# B&R Automation Studio project NAINV104C00R8L515F00 (part 20)

#### Init.st
```iecst
(** 2019-05-04 **)
PROGRAM _INIT

	(* Always Change If Project Change *)

	//Pass Address To Global Address For External Use
	//Action, State & Status
	p_McParamStat		:= ADR(eStat);
	p_McParamStatus		:= ADR(eStatus);
	p_McParamStatTxt	:= ADR(sStatTxt);

	//Alarm
	p_McParamAlmData	:= ADR(tyAlmData);

	//Output
	p_McParamFileNotFound			:= ADR(bFileNotFound);

	p_McParamCurr					:= ADR(tyMcParamCurr);

	p_McParamLFOnline				:= ADR(tyMcParamCurr.a_bLFOnline);
	p_McParamLFIPAddr				:= ADR(tyMcParamCurr.a_sLFIPAddr);

	p_McParamMcNm					:= ADR(tyMcParamCurr.sMcNm);
	p_McParamWidthAtHmPos			:= ADR(tyMcParamCurr.diWidthAtHmPosInUM);
	p_McParamWidthOffset			:= ADR(tyMcParamCurr.diWidthOffsetInUM);
	p_McParamSSaverEn				:= ADR(tyMcParamCurr.bSSaverEn);
	p_McParamSSaverTm				:= ADR(tyMcParamCurr.uiSSaverTmInSec);
	p_McParamConvInitTm				:= ADR(tyMcParamCurr.diConvInitTmInMS);
	p_McParamTranInErrDlyTm			:= ADR(tyMcParamCurr.diTranInErrDlyTmInMS);
	p_McParamTranOutErrDlyTm		:= ADR(tyMcParamCurr.diTranOutErrDlyTmInMS);
	p_McParamDefaultMcMod			:= ADR(tyMcParamCurr.usiDefaultMcMod);
	p_McParamDefaultFlippedBrd		:= ADR(tyMcParamCurr.usiDefaultFlippedBrd);
	p_McParamAutoStepEn				:= ADR(tyMcParamCurr.bAutoStepEn);
	p_McParamAWDis					:= ADR(tyMcParamCurr.bAWDis);
	p_McParamVSMEMAEn				:= ADR(tyMcParamCurr.bVSMEMAEn);
	p_McParamMnlAccDat				:= ADR(tyMcParamCurr.bMnlAccDat);
	p_McParamChgParamEn				:= ADR(tyMcParamCurr.bChgParamEn);
	p_McParamHermesRmtEn			:= ADR(tyMcParamCurr.bHermesRmtEn);
	p_McParamLang					:= ADR(tyMcParamCurr.usiLang);

	p_McParamLFEn					:= ADR(tyMcParamCurr.bLFEn);
	p_McParamLCSLFEn				:= ADR(tyMcParamCurr.bLCSLFEn);
	p_McParamLCSReqRcpEn			:= ADR(tyMcParamCurr.bLCSReqRcpEn);
	p_McParamLCSManageRcpEn			:= ADR(tyMcParamCurr.bLCSManageRcpEn);
	p_McParamLCSLiveDatEn			:= ADR(tyMcParamCurr.bLCSLiveDatEn);
	p_McParamSectionLeader			:= ADR(tyMcParamCurr.bSectionLeader);
	p_McParamUSWidthChkEn			:= ADR(tyMcParamCurr.bUSWidthChkEn);
	p_McParamDSWidthChkEn			:= ADR(tyMcParamCurr.bDSWidthChkEn);

	p_McParamConvLftSenAntiGap		:= ADR(tyMcParamCurr.tyConvLftSenAntiGapDly);
	p_McParamConvLftSenOnTm			:= ADR(tyMcParamCurr.tyConvLftSenAntiGapDly.diSigOnTm);
	p_McParamConvLftSenOffTm		:= ADR(tyMcParamCurr.tyConvLftSenAntiGapDly.diSigOffTm);
	p_McParamConvRgtSenAntiGap		:= ADR(tyMcParamCurr.tyConvRgtSenAntiGapDly);
	p_McParamConvRgtSenOnTm			:= ADR(tyMcParamCurr.tyConvRgtSenAntiGapDly.diSigOnTm);
	p_McParamConvRgtSenOffTm		:= ADR(tyMcParamCurr.tyConvRgtSenAntiGapDly.diSigOffTm);

	p_McParamUSCommMod				:= ADR(tyMcParamCurr.eUSComm);
	p_McParamUSSMEMAParam			:= ADR(tyMcParamCurr.tyUSCommSMEMA);
	p_McParamUSSMEMASelection		:= ADR(tyMcParamCurr.tyUSCommSMEMA.eSelection);
	p_McParamUBAStatSetGd			:= ADR(tyMcParamCurr.tyUSCommSMEMA.bStatSigSetGd);

	p_McParamDSCommMod				:= ADR(tyMcParamCurr.eDSComm);
	p_McParamDSSMEMAParam			:= ADR(tyMcParamCurr.tyDSCommSMEMA);
	p_McParamDSSMEMASelection		:= ADR(tyMcParamCurr.tyDSCommSMEMA.eSelection);
	p_McParamDBAStatSetGd			:= ADR(tyMcParamCurr.tyDSCommSMEMA.bStatSigSetGd);

	p_McParamStopperDis				:= ADR(tyMcParamCurr.bStopperDis);
	p_McParamStopperAtLftPos		:= ADR(tyMcParamCurr.diStopperAtLftPos);
	p_McParamStopperAtRgtPos		:= ADR(tyMcParamCurr.diStopperAtRgtPos);
	p_McParamLFLeaderMc				:= ADR(tyMcParamCurr.bLFLeaderMc);
	p_McParamLFMcIdxBeforeOven		:= ADR(tyMcParamCurr.diLFMcIdxBeforeOven);
	p_McParamLFMcIdxAfterOven		:= ADR(tyMcParamCurr.diLFMcIdxAfterOven);
	p_McParamLFMcIdxBeforeOven2		:= ADR(tyMcParamCurr.diLFMcIdxBeforeOven2);
	p_McParamLFMcIdxAfterOven2		:= ADR(tyMcParamCurr.diLFMcIdxAfterOven2);

	p_McParamClampDis				:= ADR(tyMcParamCurr.bClampDis);

	p_McParamInShutterDis			:= ADR(tyMcParamCurr.bInShutterDis);
	p_McParamOutShutterDis			:= ADR(tyMcParamCurr.bOutShutterDis);

	p_McParamNetworkMod				:= ADR(tyMcParamCurr.eNetworkMod);
	p_McParamLFSeqStayActive		:= ADR(tyMcParamCurr.bLFSeqStayActive);
	p_McParamLFBuzMute				:= ADR(tyMcParamCurr.bLFBuzMute);
	p_McParamDBAOnWOAlign			:= ADR(tyMcParamCurr.bDBAOnWOAlign);

	//InvertOnce & InvertTwice_2023_0032B01
	p_McParamUSComm2Mod				:= ADR(tyMcParamCurr.eUSComm2);
	p_McParamUSSMEMA2Param			:= ADR(tyMcParamCurr.tyUSCommSMEMA2);
	p_McParamUSSMEMA2Selection		:= ADR(tyMcParamCurr.tyUSCommSMEMA2.eSelection);
	p_McParamUBAStat2SetGd			:= ADR(tyMcParamCurr.tyUSCommSMEMA2.bStatSigSetGd);

	//process machine to inverter
	p_McParamDSComm2Mod				:= ADR(tyMcParamCurr.eDSComm2);
	p_McParamDSSMEMA2Param			:= ADR(tyMcParamCurr.tyDSCommSMEMA2);
	p_McParamDSSMEMA2Selection		:= ADR(tyMcParamCurr.tyDSCommSMEMA2.eSelection);
	p_McParamDBAStat2SetGd			:= ADR(tyMcParamCurr.tyDSCommSMEMA2.bStatSigSetGd);

	(* Always Change If Project Change *)

END_PROGRAM
```

### NtParam.typ - Change By Project
```iecst
(*2020-10-06*)
(**)
(*Action*)

TYPE
	eNtParamAction :
		(
		NtParamActIdle,
		NtParamActCreateDir,
		NtParamActRead,
		NtParamActWrite,
		NtParamActLoad,
		NtParamActSave
		);
END_TYPE

(**)
(*Data*)

TYPE
	tyNtParam : 	STRUCT
		tyDISettings : tyDigitalInputSettings := (diSafetyRlySig:=1,diEStopSig:=2,diCoverSWSig:=3,diUBA:=4,diUBAStat:=0,diDSB:=5,diConvLftSen:=7,diConvRgtSen:=8,diPressureSW:=0,diCoatingSen:=0,diThermalPrtSig:=0,diUSWidthChkSen:=0,diDSWidthChkSen:=0,diInvertHomeSen:=9,diInvertRemoteSen:=10,diInShutterOpenRS:=14,diInShutterCloseRS:=13,diOutShutterOpenRS:=16,diOutShutterCloseRS:=15,diClamp2Sen:=19,diClamp3Sen:=20,diClampRS1:=22,diUnClampRS1:=21,diClampRS2:=24,diUnClampRS2:=23,diClampRS3:=26,diUnClampRS3:=25,diUSWidthChkSen1:=0,diCoverSWSig2:=17,diSafetySigFromUS:=29,diSafetySigFromDS:=30,diUnlockCoverSigFromUS:=27,diUnlockCoverSigFromDS:=28,diCoverUnlockPB1:=31,diUBA2:=0,diUBAStat2:=0,diSPARE9:=0,diSPARE10:=0,diSPARE11:=0,diSPARE12:=0);
		tyDOSettings : tyDigitalOutputSettings := (diSafetyRlyRst:=1,diTLRed:=4,diTLAmber:=3,diTLGreen:=2,diTLBlue:=0,diTLWhite:=0,diBuz:=5,diCoatingStprRet:=0,diUSB:=8,diDBA:=9,diDBAStat:=0,diConvMtrCW:=11,diConvMtrCCW:=12,diStprUnblkCtrl:=13,diStprBlkCtrl:=14,diInvertHome:=15,diInvertRemote:=16,diInvertBrake:=17,diMtrPwrRly:=0,diClampControl:=0,diUnclampControl:=0,diInShutterOpenCtrl:=20,diInShutterCloseCtrl:=19,diOutShutterOpenCtrl:=22,diOutShutterCloseCtrl:=21,diClamp1Ctrl:=23,diUnClamp1Ctrl:=24,diClamp2Ctrl:=25,diUnClamp2Ctrl:=26,diClamp3Ctrl:=27,diUnClamp3Ctrl:=28,diTopCvrUnlckToDS:=30,diTopCvrUnlckToUS:=0,diMachineSafetySigToDS:=29,diMachineSafetySigToUS:=0,diCoverPBLED1:=31,diBypassTopCover1:=32,diSafetyTopCoverSWCoil1:=33,diUSB2:=0,diSPARE9:=0,diSPARE10:=0,diSPARE11:=0,diSPARE12:=0);
		bAWPrep : BOOL := TRUE;
		bLFPrep : BOOL := TRUE;
		bLeaderMc : BOOL := FALSE;
		bLFUsrSetPrep : BOOL := TRUE;
		diLFWidthLimit : DINT := 3000;
		bLFProdWidthChk : BOOL := TRUE;
		bLFProdWidth2Prep : BOOL := FALSE;
		bUSWidthChkPrep : BOOL := FALSE;
		bDSWidthChkPrep : BOOL := FALSE;
		bLCSLFPrep : BOOL := FALSE;
		bLCSReqRcpPrep : BOOL := FALSE;
		bLCSManageRcpPrep : BOOL := FALSE;
		bLCSLiveDatPrep : BOOL := FALSE;
		bUSExtSMEMAPrep : BOOL := TRUE;
		bDSExtSMEMAPrep : BOOL := TRUE;
		bVSMEMAPrep : BOOL := TRUE;
		bHermesPrep : BOOL := TRUE;
		bHermesRmtPrep : BOOL := TRUE;
		bUnlockCoverPrep : BOOL := FALSE;
		bUSDSMachineSafetySig : BOOL := FALSE;
		bSSaverPrep : BOOL := TRUE;
		bAutoLogoutPrep : BOOL := TRUE;
		diWidthOffsetInUM : DINT := 0;
		tyUIAWOffset : tyUILmt := (diMax:=2000,diMin:=-2000);
		sJobNo : STRING[30] := '2022-0669Q01';
		usiNtAddr : USINT := 4;
		eProjConvDir : eConvDir := ConvDirLToR;
		bProjCoatingPrep : BOOL := FALSE;
		tComLoadRstTm : TIME := T#1s; (*Common Layer Loading Time*)
		bProjDBAOnRgtSen : BOOL := FALSE;
		bProjClampPrep : BOOL := TRUE;
		eProjClampOption : eClampType := ThreeClampsWithRS;
		bProjStopperPrep : BOOL := TRUE;
		bProjInletShutPrep : BOOL := TRUE;
		bProjOutletShutPrep : BOOL := TRUE;
		bProjBypsInitConvPrep : BOOL := TRUE;
		bProjRlsNewProdPrep : BOOL := FALSE;
		sUsrFolderProgNm : STRING[15] := 'UsrFolder';
		sLibVersionProgNm : STRING[15] := 'LibVer';
		sTimeProgNm : STRING[15] := 'Time';
		sHWInfoProgNm : STRING[15] := 'HWInfo';
		sHWInfoDevice : STRING[3] := 'IF2';
		sAlmProgNm : STRING[15] := 'Alarm';
		tTLChgRcpBlinkTm : TIME := T#500ms;
		tTLErrBlinkTm : TIME := T#500ms;
		tBuzErrOnTm : TIME := T#500ms;
		tBuzErrRestTm : TIME := T#500ms;
		usiBuzErrOnCntr : USINT := 3;
		bBuzErrStopSeqEn : BOOL := FALSE;
		usiBuzErrStopSeqCntr : USINT := 3;
		tTLWarnBlinkTm : TIME := T#500ms;
		tBuzWarnOnTm : TIME := T#500ms;
		tBuzWarnRestTm : TIME := T#5s;
		usiBuzWarnOnCntr : USINT := 3;
		bBuzWarnStopSeqEn : BOOL := FALSE;
		usiBuzWarnStopSeqCntr : USINT := 3;
		tTLWarn1BlinkTm : TIME := T#500ms;
		tBuzWarn1OnTm : TIME := T#500ms;
		tBuzWarn1RestTm : TIME := T#5s;
		usiBuzWarn1OnCntr : USINT := 3;
		bBuzWarn1StopSeqEn : BOOL := FALSE;
		usiBuzWarn1StopSeqCntr : USINT := 3;
		tTLWarn2BlinkTm : TIME := T#500ms;
		tBuzWarn2OnTm : TIME := T#500ms;
		tBuzWarn2RestTm : TIME := T#5s;
		usiBuzWarn2OnCntr : USINT := 3;
		bBuzWarn2StopSeqEn : BOOL := FALSE;
		usiBuzWarn2StopSeqCntr : USINT := 3;
		tTLWarn3BlinkTm : TIME := T#500ms;
		tBuzWarn3OnTm : TIME := T#500ms;
		tBuzWarn3RestTm : TIME := T#5s;
		usiBuzWarn3OnCntr : USINT := 3;
		bBuzWarn3StopSeqEn : BOOL := FALSE;
		usiBuzWarn3StopSeqCntr : USINT := 3;
		tTLWarn4BlinkTm : TIME := T#500ms;
		tBuzWarn4OnTm : TIME := T#500ms;
		tBuzWarn4RestTm : TIME := T#5s;
		usiBuzWarn4OnCntr : USINT := 3;
		bBuzWarn4StopSeqEn : BOOL := FALSE;
		usiBuzWarn4StopSeqCntr : USINT := 3;
		tTLWarn5BlinkTm : TIME := T#500ms;
		tBuzWarn5OnTm : TIME := T#500ms;
		tBuzWarn5RestTm : TIME := T#5s;
		usiBuzWarn5OnCntr : USINT := 3;
		bBuzWarn5StopSeqEn : BOOL := FALSE;
		usiBuzWarn5StopSeqCntr : USINT := 3;
		tBuzAlertOnTm : TIME := T#500ms;
		tBuzAlertRestTm : TIME := T#5s;
		usiBuzAlertOnCntr : USINT := 3;
		bBuzAlertStopSeqEn : BOOL := FALSE;
		usiBuzAlertStopSeqCntr : USINT := 3;
		tTLBlueBlinkTm : TIME := T#500ms;
		tTLAmberBlinkTm : TIME := T#500ms;
		tTLWhiteBlinkTm : TIME := T#500ms;
		tTLRedBlinkTm : TIME := T#500ms;
		tTLGreenBlinkTm : TIME := T#500ms;
		eTLBuzMode : eTLBuzMod := TLBuzModNutek;
		udiAlmFileKeepDay : UDINT := 30;
		sProdRcpProgNm : STRING[15] := 'ProdRcp';
		sProdRcpListFileNm : STRING[80] := 'ProductRecipeList.dat';
		sProdRcpSingleFileNm : STRING[80] := 'ProductRecipe.dat';
		sMpProdRcpProgNm : STRING[15] := 'MpProdRcp';
		sMpProdRcpFileNm : STRING[255] := 'MpProductRecipe.xml';
		sMpProdRcpPVNm : STRING[100] := 'MpProdRcp:a_tyMpProdRcp1';
		sMcParamProgNm : STRING[15] := 'McParam';
		sMcParamFileNm : STRING[80] := 'MachineParameter.dat';
		sUsrMgmtProgNm : STRING[15] := 'UsrMgmt';
		sUSSMEMAProgNm : STRING[15] := 'USSMEMA';
		tUSSMEMARstDlyTm : TIME := T#0s;
		tUSSMEMASigInChkTm : TIME := T#100ms;
		sDSSMEMAProgNm : STRING[15] := 'DSSMEMA';
		tDSSMEMARstDlyTm : TIME := T#0s;
		tDSSMEMASigInChkTm : TIME := T#100ms;
		sConvProgNm : STRING[15] := 'Conv';
		bConvOnDirMod : BOOL := FALSE;
		tConvMtrOffDlyTm : TIME := T#0s;
		diConvFwdDlyTm : DINT := 5000;
		diConvRevDlyTm : DINT := 5000;
		sStopperProgNm : STRING[15] := 'Stopper';
		bStopperTwoCtrlIn : BOOL := TRUE;
		tStopperExtDlyTm : TIME := T#1s;
		tStopperRetDlyTm : TIME := T#1s;
		sClampProgNm : STRING[15] := 'Clamp';
		bClampTwoCtrlIn : BOOL := TRUE;
		tClampExtDlyTm : TIME := T#1s;
		tClampRetDlyTm : TIME := T#1s;
		sInShutterProgNm : STRING[15] := 'Inlet Shutter';
		bInShutterTwoCtrlIn : BOOL := TRUE;
		tInShutterExtTO : TIME := T#20s;
		tInShutterRetTO : TIME := T#20s;
		sOutShutterProgNm : STRING[15] := 'Outlet Shutter';
		bOutShutterTwoCtrlIn : BOOL := TRUE;
		tOutShutterExtTO : TIME := T#20s;
		tOutShutterRetTO : TIME := T#20s;
		sClamp1ProgNm : STRING[15] := 'Clamp1'; (*c*)
		bClamp1TwoCtrlIn : BOOL := TRUE;
		tClamp1ExtTO : TIME := T#20s;
		tClamp1RetTO : TIME := T#20s;
		sClamp2ProgNm : STRING[15] := 'Clamp2';
		bClamp2TwoCtrlIn : BOOL := TRUE;
		tClamp2ExtTO : TIME := T#20s;
		tClamp2RetTO : TIME := T#20s;
		sClamp3ProgNm : STRING[15] := 'Clamp3';
		bClamp3TwoCtrlIn : BOOL := TRUE;
		tClamp3ExtTO : TIME := T#20s;
		tClamp3RetTO : TIME := T#20s;
		diMotorOnDlyTm : DINT := 500;
		diMotorOffDlyTm : DINT := 500;
		diBrakeOnDlyTm : DINT := 0;
		diBrakeOffDlyTm : DINT := 500;
		diTimeOut : DINT := 10000;
		sAWProgNm : STRING[15] := 'AW';
		sAWDevice : STRING[3] := 'IF7';
		usiAWNode : USINT := 16;
		bAWDir : BOOL := FALSE;
		bAWDirBl : BOOL := FALSE;
		diAWPitchInUM : DINT := 3000;
		diAWMovBlDistInUM : DINT := 3000;
		tyAWParamInHm : tyMotionCANParamInHm := (diStartVelInUMPS:=15000,diAcc:=25);
		tyAWParamInConvert : tyMotionCANParamInConvert := (diPitchInUM:=3000,diPulsePerRev:=1280000); (*estun 1048576 *)
		tyAWParam : tyMotionParam := (diAccInMS:=500,diDecInMS:=500,diAutoSpdInUMPS:=15000);
		tyAWTuning : tyMotionCANTuning := (diAsdaA2Inertia:=63,diAsdaA2PosLoopGain:=53,diAsdaA2PosFFGain:=50,diAsdaA2SpdLoopGain:=213,diAsdaA2SpdIntegral:=34,diAsdaA2LowPassFltr:=49,diAsdaA2AntiInterGain:=24,diAsdaA2FirstTorqueCmd:=300,diPronetInertia:=100,diPronetRealTimeAutoAdjSet:=0,diPronetPosLoopGain:=40,diPronetSpdLoopGain:=250,diPronetSpdIntegral:=200,diPronetTorqueFilter:=100,diPronetPosFeedForward:=0,diPronetLowSpeedTestFiltering:=0,diPronetStopMode:=5);
		eAWServoMotorType : eServoMotorType := DeltaAsdaA2; (*Selection of  Motor Brand*)
		sInvertProgNm : STRING[15] := 'Invert';
		sInvertDevice : STRING[3] := 'IF7';
		usiInvertNode : USINT := 17;
		bInvertDir : BOOL := TRUE;
		tyInvertParamInHm : tyMotionCANParamInHm := (diStartVelInUMPS:=25000,diAcc:=25);
		tyInvertParamInConvert : tyMotionCANParamInConvert;
		tyInvertParam : tyMotionParam := (diAccInMS:=500,diDecInMS:=500,diAutoSpdInUMPS:=50000);
		tyInvertTuning : tyMotionCANTuning := (diAsdaA2Inertia:=211,diAsdaA2PosLoopGain:=150,diAsdaA2PosFFGain:=50,diAsdaA2SpdLoopGain:=81,diAsdaA2SpdIntegral:=13,diAsdaA2LowPassFltr:=128,diAsdaA2AntiInterGain:=13,diAsdaA2FirstTorqueCmd:=300);
		eInvertServoMotorType : eServoMotorType := DeltaAsdaA2; (*Selection of  Motor Brand*)
		sDIProgNm : STRING[15] := 'DInput';
		sMcProgNm : STRING[15] := 'Machine';
		sHermesProgNm : STRING[15] := 'Hermes';
		sHermesRetainFileNm : STRING[80] := 'Hermes.dat';
		sHermesConfigFileNm : STRING[80] := 'Hermes.dat';
		sUSHermesProgNm : STRING[15] := 'USHermes';
		udiUSHermesFileKeepDay : UDINT := 7;
		udiUSHermesAliveTmInSec : UDINT := 5;
		tUSHermesConnTO : TIME := T#30s;
		sUSHermes2ProgNm : STRING[15] := 'USHermes';
		udiUSHermes2FileKeepDay : UDINT := 7;
		udiUSHermes2AliveTmInSec : UDINT := 5;
		tUSHermes2ConnTO : TIME := T#30s;
		sDSHermesProgNm : STRING[15] := 'DSHermes';
		udiDSHermesFileKeepDay : UDINT := 7;
		udiDSHermesAliveTmInSec : UDINT := 5;
		tDSHermesConnTO : TIME := T#30s;
		sDSHermes2ProgNm : STRING[15] := 'DSHermes';
		udiDSHermes2FileKeepDay : UDINT := 7;
		udiDSHermes2AliveTmInSec : UDINT := 5;
		tDSHermes2ConnTO : TIME := T#30s;
		sRmtHermesProgNm : STRING[15] := 'RmtHermes';
		sRmtHermesConfigFileNm : STRING[80] := 'RmtHermes.dat';
		udiRmtHermesFileKeepDay : UDINT := 7;
		udiRmtHermesAliveTmInSec : UDINT := 5;
		udiRmtHermesSndBffrSize : UDINT := 65536;
		udiRmtHermesRcvBffrSize : UDINT := 65536;
		sOpsAWProgNm : STRING[15] := 'OpsAW';
		sOpsInitConvProgNm : STRING[15] := 'Ops InitConv';
		sOpsInitPneuProgNm : STRING[15] := 'Ops InitPneu';
		sOpsConvProgNm : STRING[15] := 'Ops Conv';
		sOpsPneuProgNm : STRING[15] := 'Ops Pneu';
		sConvBffrProgNm : STRING[15] := 'ConvBuffer';
		sConvBffrFileNm : STRING[80] := 'ConvBuffer.dat';
		iConvBffrIdx : INT := 1;
		sLFLeaderProgNm : STRING[15] := 'Leader';
		tLFLeaderOnlineChkDlyTm : TIME := T#30s;
		tLFLeaderSetTmOffDlyTm : TIME := T#10s;
		sLFFollowerProgNm : STRING[15] := 'Follower';
		sFollower1ProgNm : STRING[15] := 'Follower1';
		tLFFollowerOnlineChkDlyTm : TIME := T#30s;
		sLCSProgNm : STRING[15] := 'LCS';
		sLCSMngRcpProgNm : STRING[15] := 'LCSMngRcp';
		sLCSLFProgNm : STRING[15] := 'LCSLF';
		tyProdRcpWidthLmt : tyUILmt := (diMax:=460000,diMin:=50000);
		tyProdRcpMcModLmt : tyUILmt := (diMax:=3,diMin:=0);
		tyProdRcpFlippedBrdLmt : tyUILmt := (diMax:=2,diMin:=0);
		tyUISSaverTm : tyUILmt := (diMax:=1800,diMin:=10);
		tyUIConvInitTm : tyUILmt := (diMax:=60000,diMin:=5000);
		tyUITranInErrDlyTm : tyUILmt := (diMax:=120000,diMin:=1000);
		tyUITranOutErrDlyTm : tyUILmt := (diMax:=120000,diMin:=1000);
		tyUIHermesSndAliveTm : tyUILmt := (diMax:=1800000,diMin:=5000);
		tyUIHermesLnID : tyUILmt := (diMax:=1000,diMin:=1);
		tyUIAntiGapSenOnTm : tyUILmt := (diMax:=5000,diMin:=0);
		tyUIAntiGapSenOffTm : tyUILmt := (diMax:=5000,diMin:=0);
		tyUILFIndexBeforeOven : tyUILmt := (diMax:=50,diMin:=1);
		tyUILFIndexAfterOven : tyUILmt := (diMax:=50,diMin:=1);
		tyUIAWTargetPos : tyUILmt := (diMax:=460000,diMin:=-3000);
		tyUIAWStepSize : tyUILmt := (diMax:=460000,diMin:=-460000);
		tyUIAWNomSpd : tyUILmt := (diMax:=15000,diMin:=5000);
		tyUIAWSlwSpd : tyUILmt := (diMax:=15000,diMin:=5000);
		tyUIInvertTargetPos : tyUILmt := (diMax:=110000,diMin:=-15000);
		tyUIInvertStepSize : tyUILmt := (diMax:=110000,diMin:=-110000);
		tyUIInvertNomSpd : tyUILmt := (diMax:=100000,diMin:=5000);
		tyUIInvertSlwSpd : tyUILmt := (diMax:=100000,diMin:=5000);
		tyUIHermesHostPort : tyUILmt := (diMax:=65535,diMin:=0);
		tyUIHermesSvrPort : tyUILmt := (diMax:=65535,diMin:=0);
		tyUIAutoLogoutTm : tyUILmt := (diMax:=1800000,diMin:=60000);
		tyNetworkMode : tyUILmt := (diMax:=1,diMin:=0);
		bUIConvDirRL : BOOL := FALSE;
		sMpNtParamFileNm : STRING[255] := 'NutekParameter.xml';
		sMpNtParamPVNm : STRING[100] := 'NtParam:tyMpNtParamCurr1';
		sUIDefaultLoginNm : STRING[30] := '';
		sUIDefaultLoginPw : STRING[30] := '';
		bProjInvertOncePrep : BOOL := TRUE;
		bProjInvertTwicePrep : BOOL := TRUE;
		bUSExtSMEMA2Prep : BOOL := TRUE;
		sUSSMEMA2ProgNm : STRING[15] := 'USSMEMA2';
		tUSSMEMA2RstDlyTm : TIME := T#0s;
		tUSSMEMA2SigInChkTm : TIME := T#100ms;
		eProjRtrnBrdConvDir : eConvDir := ConvDirRToR;
		bChinesePrep : BOOL := FALSE;
		bGemanPrep : BOOL := FALSE;
		bHermesSvyPrep : BOOL := TRUE; (*Supervisory Hermes Preparation*)
		bHermesSvyFirstMcInTheLine : BOOL := FALSE; (*Turn On this for Loader / Destacker Only. Other type of machine turns off.*)
		bHermesSvyQueryBoardInfo : BOOL := FALSE;
		sDSHermesRetainFileNm : STRING[80] := 'BoardData.dat';
		iInput : INT;
		iOutput : INT;
	END_STRUCT;
END_TYPE

(**)

TYPE
	tyUILmt : 	STRUCT
		diMax : DINT;
		diMin : DINT;
	END_STRUCT;
END_TYPE
```

### NtParam.var - Change By Project
```iecst
(*2020-10-06*)
(**)
(*Action & State & Status*)
VAR
	p_NtParamStat : UDINT;
	p_NtParamStatus : UDINT;
	p_NtParamStatTxt : UDINT;
END_VAR
(**)
(*Alarm*)
VAR
	p_NtParamAlmData : UDINT;
END_VAR
(**)
(*Output*)
VAR
	p_NtParamFileNotFound : UDINT;
END_VAR
(**)
VAR
	p_NtParamCurr : UDINT;
	p_NtParamDISettings : UDINT;
	p_NtParamDOSettings : UDINT;
	p_NtParamAWPrep : UDINT;
	p_NtParamLFPrep : UDINT;
	p_NtParamLeaderMc : UDINT;
	p_NtParamLFUsrSetPrep : UDINT;
	p_NtParamLFWidthLimit : UDINT;
	p_NtParamLFProdWidthChk : UDINT;
	p_NtParamUSWidthChkPrep : UDINT;
	p_NtParamDSWidthChkPrep : UDINT;
	p_NtParamLCSLFPrep : UDINT;
	p_NtParamLCSReqRcpPrep : UDINT;
	p_NtParamLCSManageRcpPrep : UDINT;
	p_NtParamLCSLiveDatPrep : UDINT;
	p_NtParamUSExtSMEMAPrep : UDINT;
	p_NtParamDSExtSMEMAPrep : UDINT;
	p_NtParamVSMEMAPrep : UDINT;
	p_NtParamHermesPrep : UDINT;
	p_NtParamHermesRmtPrep : UDINT;
	p_NtParamSSaverPrep : UDINT;
	p_NtParamWidthOffset : UDINT;
	p_NtParamJobNo : UDINT;
	p_NtParamNtAddr : UDINT;
END_VAR
(**)
VAR
	p_NtParamProjConvDir : UDINT;
	p_NtParamProjBypsInitConvPrep : UDINT;
	p_NtParamProjCoatingPrep : UDINT;
	p_NtParamProjClampPrep : UDINT;
	p_NtParamProjClampOption : UDINT;
	p_NtParamProjStopperPrep : UDINT;
	p_NtParamProjInletShutPrep : UDINT;
	p_NtParamProjOutletShutPrep : UDINT;
	p_NtParamProjRlsNewProdPrep : UDINT;
END_VAR
(**)
VAR
	p_NtParamUsrFolderProgNm : UDINT;
END_VAR
(**)
VAR
	p_NtParamLibVersionProgNm : UDINT;
END_VAR
(**)
VAR
	p_NtParamTimeProgNm : UDINT;
END_VAR
(**)
VAR
	p_NtParamHWInfoProgNm : UDINT;
	p_NtParamHWInfoDevice : UDINT;
END_VAR
(**)
VAR
	p_NtParamTLChgRcpBlinkTm : UDINT;
	p_NtParamTLErrBlinkTm : UDINT;
	p_NtParamBuzErrOnTm : UDINT;
	p_NtParamBuzErrRestTm : UDINT;
	p_NtParamBuzErrOnCntr : UDINT;
	p_NtParamBuzErrStopSeqEn : UDINT;
	p_NtParamBuzErrStopSeqCntr : UDINT;
END_VAR
(**)
VAR
	p_NtParamTLWarnBlinkTm : UDINT;
	p_NtParamBuzWarnOnTm : UDINT;
	p_NtParamBuzWarnRestTm : UDINT;
	p_NtParamBuzWarnOnCntr : UDINT;
	p_NtParamBuzWarnStopSeqEn : UDINT;
	p_NtParamBuzWarnStopSeqCntr : UDINT;
END_VAR
(**)
VAR
	p_NtParamTLWarn1BlinkTm : UDINT;
	p_NtParamBuzWarn1OnTm : UDINT;
	p_NtParamBuzWarn1RestTm : UDINT;
	p_NtParamBuzWarn1OnCntr : UDINT;
	p_NtParamBuzWarn1StopSeqEn : UDINT;
	p_NtParamBuzWarn1StopSeqCntr : UDINT;
END_VAR
(**)
VAR
	p_NtParamTLWarn2BlinkTm : UDINT;
	p_NtParamBuzWarn2OnTm : UDINT;
	p_NtParamBuzWarn2RestTm : UDINT;
	p_NtParamBuzWarn2OnCntr : UDINT;
	p_NtParamBuzWarn2StopSeqEn : UDINT;
	p_NtParamBuzWarn2StopSeqCntr : UDINT;
END_VAR
(**)
VAR
	p_NtParamTLWarn3BlinkTm : UDINT;
	p_NtParamBuzWarn3OnTm : UDINT;
	p_NtParamBuzWarn3RestTm : UDINT;
	p_NtParamBuzWarn3OnCntr : UDINT;
	p_NtParamBuzWarn3StopSeqEn : UDINT;
	p_NtParamBuzWarn3StopSeqCntr : UDINT;
END_VAR
(**)
VAR
	p_NtParamTLWarn4BlinkTm : UDINT;
	p_NtParamBuzWarn4OnTm : UDINT;
	p_NtParamBuzWarn4RestTm : UDINT;
	p_NtParamBuzWarn4OnCntr : UDINT;
	p_NtParamBuzWarn4StopSeqEn : UDINT;
	p_NtParamBuzWarn4StopSeqCntr : UDINT;
END_VAR
(**)
VAR
	p_NtParamTLWarn5BlinkTm : UDINT;
	p_NtParamBuzWarn5OnTm : UDINT;
	p_NtParamBuzWarn5RestTm : UDINT;
	p_NtParamBuzWarn5OnCntr : UDINT;
	p_NtParamBuzWarn5StopSeqEn : UDINT;
	p_NtParamBuzWarn5StopSeqCntr : UDINT;
END_VAR
(**)
VAR
	p_NtParamBuzAlertOnTm : UDINT;
	p_NtParamBuzAlertRestTm : UDINT;
	p_NtParamBuzAlertOnCntr : UDINT;
	p_NtParamBuzAlertStopSeqEn : UDINT;
	p_NtParamBuzAlertStopSeqCntr : UDINT;
END_VAR
(**)
VAR
	p_NtParamTLBlueBlinkTm : UDINT;
	p_NtParamTLAmberBlinkTm : UDINT;
	p_NtParamTLWhiteBlinkTm : UDINT;
	p_NtParamTLRedBlinkTm : UDINT;
	p_NtParamTLGreenBlinkTm : UDINT;
END_VAR
(**)
VAR
	p_NtParamTLBuzErrBlinkTm : UDINT;
	p_NtParamTLBuzChgRcpBlinkTm : UDINT;
	p_NtParamTLBuzWarnBlinkTm : UDINT;
	p_NtParamTLBuzWarnRestTm : UDINT;
	p_NtParamTLBuzWarnOnTm : UDINT;
	p_NtParamTLBuzWarn1BlinkTm : UDINT;
	p_NtParamTLBuzWarn1RestTm : UDINT;
	p_NtParamTLBuzWarn1OnTm : UDINT;
	p_NtParamTLBuzWarn2BlinkTm : UDINT;
	p_NtParamTLBuzWarn2RestTm : UDINT;
	p_NtParamTLBuzWarn2OnTm : UDINT;
	p_NtParamTLBuzWarn3BlinkTm : UDINT;
	p_NtParamTLBuzWarn3RestTm : UDINT;
	p_NtParamTLBuzWarn3OnTm : UDINT;
	p_NtParamTLBuzWarn4BlinkTm : UDINT;
	p_NtParamTLBuzWarn4RestTm : UDINT;
	p_NtParamTLBuzWarn4OnTm : UDINT;
	p_NtParamTLBuzWarn5BlinkTm : UDINT;
	p_NtParamTLBuzWarn5RestTm : UDINT;
	p_NtParamTLBuzWarn5OnTm : UDINT;
	p_NtParamTLBuzMode : UDINT;
END_VAR
(**)
VAR
	p_NtParamAlmProgNm : UDINT;
	p_NtParamAlmFileKeepDay : UDINT;
END_VAR
(**)
VAR
	p_NtParamProdRcpProgNm : UDINT;
	p_NtParamProdRcpListFileNm : UDINT;
	p_NtParamProdRcpSingleFileNm : UDINT;
END_VAR
(**)
VAR
	p_NtParamMpProdRcpProgNm : UDINT;
	p_NtParamMpProdRcpFileNm : UDINT;
	p_NtParamMpProdRcpPVNm : UDINT;
END_VAR
(**)
VAR
	p_NtParamMcParamProgNm : UDINT;
	p_NtParamMcParamFileNm : UDINT;
END_VAR
(**)
VAR
	p_NtParamUsrMgmtProgNm : UDINT;
END_VAR
(**)
VAR
	p_NtParamUSSMEMAProgNm : UDINT;
	p_NtParamUSSMEMARstDlyTm : UDINT;
	p_NtParamUSSMEMASigInChkTm : UDINT;
END_VAR
(**)
VAR
	p_NtParamDSSMEMAProgNm : UDINT;
	p_NtParamDSSMEMARstDlyTm : UDINT;
	p_NtParamDSSMEMASigInChkTm : UDINT;
END_VAR
(**)
VAR
	p_NtParamConvProgNm : UDINT;
	p_NtParamConvOnDirMod : UDINT;
	p_NtParamConvMtrOffDlyTm : UDINT;
	p_NtParamConvFwdDlyTm : UDINT;
	p_NtParamConvRevDlyTm : UDINT;
END_VAR
(**)
VAR
	p_NtParamStopperProgNm : UDINT;
	p_NtParamStopperTwoCtrlIn : UDINT;
	p_NtParamStopperExtDlyTm : UDINT;
	p_NtParamStopperRetDlyTm : UDINT;
END_VAR
(**)
VAR
	p_NtParamClampProgNm : UDINT;
	p_NtParamClampTwoCtrlIn : UDINT;
	p_NtParamClampExtDlyTm : UDINT;
	p_NtParamClampRetDlyTm : UDINT;
END_VAR
(**)
VAR
	p_NtParamInShutterProgNm : UDINT;
	p_NtParamInShutterTwoCtrlIn : UDINT;
	p_NtParamInShutterExtTO : UDINT;
	p_NtParamInShutterRetTO : UDINT;
END_VAR
(**)
VAR
	p_NtParamOutShutterProgNm : UDINT;
	p_NtParamOutShutterTwoCtrlIn : UDINT;
	p_NtParamOutShutterExtTO : UDINT;
	p_NtParamOutShutterRetTO : UDINT;
END_VAR
(**)
VAR
	p_NtParamClamp1ProgNm : UDINT;
	p_NtParamClamp1TwoCtrlIn : UDINT;
	p_NtParamClamp1ExtTO : UDINT;
	p_NtParamClamp1RetTO : UDINT;
END_VAR
(**)
VAR
	p_NtParamClamp2ProgNm : UDINT;
	p_NtParamClamp2TwoCtrlIn : UDINT;
	p_NtParamClamp2ExtTO : UDINT;
	p_NtParamClamp2RetTO : UDINT;
END_VAR
(**)
VAR
	p_NtParamClamp3ProgNm : UDINT;
	p_NtParamClamp3TwoCtrlIn : UDINT;
	p_NtParamClamp3ExtTO : UDINT;
	p_NtParamClamp3RetTO : UDINT;
END_VAR
(**)
VAR
	p_NtParamMotorOnDlyTm : UDINT;
	p_NtParamMotorOffDlyTm : UDINT;
	p_NtParamBrakeOnDlyTm : UDINT;
	p_NtParamBrakeOffDlyTm : UDINT;
	p_NtParamTimeOut : UDINT;
END_VAR
(**)
VAR
	p_NtParamAWProgNm : UDINT;
	p_NtParamAWDevice : UDINT;
	p_NtParamAWNode : UDINT;
	p_NtParamAWDir : UDINT;
	p_NtParamAWDirBl : UDINT;
	p_NtParamAWPitchInUM : UDINT;
	p_NtParamAWMovBlDistInUM : UDINT;
	p_NtParamAWParamInHm : UDINT;
	p_NtParamAWParamInConvert : UDINT;
	p_NtParamAWParam : UDINT;
	p_NtParamAWAcc : UDINT;
	p_NtParamAWDec : UDINT;
	p_NtParamAWAutoSpd : UDINT;
	p_NtParamAWTuning : UDINT;
	p_NtParamAWMotorType : UDINT;
END_VAR
(**)
VAR
	p_NtParamInvertProgNm : UDINT;
	p_NtParamInvertDevice : UDINT;
	p_NtParamInvertNode : UDINT;
	p_NtParamInvertDir : UDINT;
	p_NtParamInvertParamInHm : UDINT;
	p_NtParamInvertParamInConvert : UDINT;
	p_NtParamInvertParam : UDINT;
	p_NtParamInvertAcc : UDINT;
	p_NtParamInvertDec : UDINT;
	p_NtParamInvertAutoSpd : UDINT;
	p_NtParamInvertTuning : UDINT;
	p_NtParamInvertMotorType : UDINT;
END_VAR
(**)
VAR
	p_NtParamDInputProgNm : UDINT;
END_VAR
(**)
VAR
	p_NtParamMcProgNm : UDINT;
END_VAR
(**)
VAR
	p_NtParamHermesProgNm : UDINT;
	p_NtParamHermesRetainFileNm : UDINT;
	p_NtParamHermesConfigFileNm : UDINT;
END_VAR
(**)
VAR
	p_NtParamUSHermesProgNm : UDINT;
	p_NtParamUSHermesFileKeepDay : UDINT;
	p_NtParamUSHermesAliveTmInSec : UDINT;
	p_NtParamUSHermesConnTO : UDINT;
END_VAR
(**)
VAR
	p_NtParamDSHermesProgNm : UDINT;
	p_NtParamDSHermesFileKeepDay : UDINT;
	p_NtParamDSHermesAliveTmInSec : UDINT;
	p_NtParamDSHermesConnTO : UDINT;
END_VAR
(*US Hermes 2*)
VAR
	p_NtParamUSHermes2ProgNm : UDINT;
	p_NtParamUSHermes2FileKeepDay : UDINT;
	p_NtParamUSHermes2AliveTmInSec : UDINT;
	p_NtParamUSHermes2ConnTO : UDINT;
END_VAR
(*DS Hermes2*)
VAR
	p_NtParamDSHermes2ProgNm : UDINT;
	p_NtParamDSHermes2FileKeepDay : UDINT;
	p_NtParamDSHermes2AliveTmInSec : UDINT;
	p_NtParamDSHermes2ConnTO : UDINT;
END_VAR
(**)
VAR
	p_NtParamRmtHermesProgNm : UDINT;
	p_NtParamRmtHermesConfigFileNm : UDINT;
	p_NtParamRmtHermesFileKeepDay : UDINT;
	p_NtParamRmtHermesAliveTmInSec : UDINT;
	p_NtParamRmtHermesSndBffrSize : UDINT;
	p_NtParamRmtHermesRcvBffrSize : UDINT;
END_VAR
(**)
VAR
	p_NtParamOpsAWProgNm : UDINT;
	p_NtParamOpsInitConvProgNm : UDINT;
	p_NtParamOpsInitPneuProgNm : UDINT;
	p_NtParamOpsConvProgNm : UDINT;
	p_NtParamOpsPneuProgNm : UDINT;
END_VAR
(**)
VAR
	p_NtParamConvBffrProgNm : UDINT;
	p_NtParamConvBffrFileNm : UDINT;
	p_NtParamConvBffrIdx : UDINT;
END_VAR
(**)
VAR
	p_NtParamLFLeaderProgNm : UDINT;
	p_NtParamLFLeaderOnlineChkDlyTm : UDINT;
	p_NtParamLFLeaderSetTmOffDlyTm : UDINT;
END_VAR
(**)
VAR
	p_NtParamLFFollowerProgNm : UDINT;
END_VAR
(**)
VAR
	p_NtParamFollower1ProgNm : UDINT;
END_VAR
(**)
VAR
	p_NtParamLCSProgNm : UDINT;
END_VAR
(**)
VAR
	p_NtParamLCSMngRcpProgNm : UDINT;
END_VAR
(**)
VAR
	p_NtParamLCSLFProgNm : UDINT;
END_VAR
(**)
VAR
	p_NtParamProdRcpMinWidth : UDINT;
	p_NtParamProdRcpMaxWidth : UDINT;
	p_NtParamProdRcpMinMcMod : UDINT;
	p_NtParamProdRcpMaxMcMod : UDINT;
	p_NtParamProdRcpMinFlippedBrd : UDINT;
	p_NtParamProdRcpMaxFlippedBrd : UDINT;
END_VAR
(**)
VAR
	p_NtParamUIConvDirRL : UDINT;
	p_NtParamProjDBAOnRgtSen : UDINT;
END_VAR
(**)
VAR
	p_NtParamLFWidth2Prep : UDINT;
	p_NtParamLFFllowerOnlineChkDlyTm : UDINT;
END_VAR
(**)
VAR
	p_NTParamUnlockCovPrep : UDINT;
	p_NTParamMachineSafetySig : UDINT;
END_VAR
(**)
VAR
	p_NtParamProjInvertOncePrep : UDINT;
	p_NtParamProjInvertTwicePrep : UDINT;
	p_NtParamUSExtSMEMA2Prep : UDINT;
	p_NtParamUSSMEMA2ProgNm : UDINT;
	p_NtParamUSSMEMA2RstDlyTm : UDINT;
	p_NtParamUSSMEMA2SigInChkTm : UDINT;
	p_NtParamProjRtrnBrdConvDir : UDINT;
END_VAR
(**)
VAR
	p_NtParamProjChinesePrep : UDINT;
	p_NtParamProjGermanPrep : UDINT;
END_VAR
(* *)
VAR
	p_NtParamHermesInput : UDINT;
	p_NtParamHermesOutput : UDINT;
END_VAR
(* *)
VAR
	p_NtParamHermesSvyPrep : UDINT;
	p_NtParamDSHermesRetainFileNm : UDINT;
END_VAR
```

### Program Logical/NtParam/NtParam (IEC)

#### InputRef.var
```iecst
(*2020-07-27*)
(**)
(*General*)
VAR
	p_eAct : REFERENCE TO eNtParamAction;
	p_udiRstErr : REFERENCE TO UDINT;
END_VAR
(**)
(*Configuration*)
VAR
	p_sFileName : REFERENCE TO STRING[80];
	p_sProgNm : REFERENCE TO STRING[15];
	p_sFileName1 : REFERENCE TO STRING[80];
	p_sPVName : REFERENCE TO STRING[80];
	p_tyMpNtParamMpLink : REFERENCE TO MpComIdentType;
END_VAR
```

#### InputRef_Link.var
```iecst
(*2019-03-25*)
(**)
VAR
	p_bLinkStartupRun : REFERENCE TO BOOL;
END_VAR
```

#### Local.var
```iecst
(*2020-07-27*)
(**)
(*Local Action, State & Status*)
VAR
	eAct : eNtParamAction := NtParamActIdle;
	eStat : eNtParamAction := NtParamActIdle;
	eStatus : eFBStatus := Idle;
	udiStatus : UDINT := 0;
	sStatTxt : STRING[200] := '';
	a_sStatText : ARRAY[0..50] OF STRING[200] := ['Idling','Creating Directory','Reading Files','Writing Files','Loading Data From XML','Saving Data To XML',45('')];
END_VAR
(**)
(*Local Alarm*)
VAR
	tyAlmData : tyAlmDat;
	a_tyAlmText : ARRAY[10000..10099] OF tyAlmTxt := [(sAlmText:='Create User Directory Error',sRcyText:='Unable To Create User Directory. Please Contact Nutek For A Possible Solution'),(sAlmText:='Create Nutek Parameter Directory Error',sRcyText:='Unable To Create Nutek Parameter Directory. Please Contact Nutek For A Possible Solution'),(sAlmText:='File Open Error While Writing',sRcyText:='An Error Was Encountered While Trying To Open File. Please Contact Nutek For A Possible Solution.'),(sAlmText:='File Create Error While Writing',sRcyText:='An Error Was Encountered While Trying To Create File. Please Contact Nutek For A Possible Solution.'),(sAlmText:='File Write Error',sRcyText:='An Error Was Encountered While Trying To Write File. Please Contact Nutek For A Possible Solution.'),(sAlmText:='File Close Error While Writing',sRcyText:='An Error Was Encountered While Trying To Close File. Please Contact Nutek For A Possible Solution.'),(sAlmText:='File Open Error While Reading',sRcyText:='An Error Was Encountered While Trying To Open File. Please Contact Nutek For A Possible Solution.'),(sAlmText:='File Read Error',sRcyText:='An Error Was Encountered While Trying To Read File. Please Contact Nutek For A Possible Solution.'),(sAlmText:='File Close Error While Reading',sRcyText:='An Error Was Encountered While Trying To Close File. Please Contact Nutek For A Possible Solution.'),(sAlmText:='Directory Does Not Exist While Writing',sRcyText:='The Directory Does Not Exist.Please Contact Nutek For A Possible Solution.'),(sAlmText:='MpRecipeRegPar Error While Loading',sRcyText:='Unable To Register Parameter. Please Contact Nutek For A Possible Solution'),(sAlmText:='MpRecipeXml Error While Loading',sRcyText:='Unable To Handle Recipe In Xml. Please Contact Nutek For A Possible Solution'),(sAlmText:='MpReipeRegPar Error While Saving',sRcyText:='Unable To Register Parameter. Please Contact Nutek For A Possible Solution'),(sAlmText:='MpRecipeXml Error While Saving',sRcyText:='Unable To Handle Recipe In Xml. Please Contact Nutek For A Possible Solution'),(sAlmText:='Create Nutek Parameter Xml Directory Error',sRcyText:='Unable To Create Nutek Parameter Xml Directory. Please Contact Nutek For A Possible Solution'),85((0))];
END_VAR
(**)
(*Local Output*)
VAR
	tyNtParamCurr : tyNtParam;
	tyMpNtParamCurr1 : tyNtParam;
	bFileNotFound : BOOL;
END_VAR
(**)
(*Local Input*)
VAR
	udiRstErr : UDINT := 0;
	sFileName : STRING[80] := 'NutekParameter.dat';
	sProgNm : STRING[15] := 'NtParam';
	sFileName1 : STRING[80] := 'NutekParameter.xml';
	sPVName : STRING[100] := 'NtParam:tyMpNtParamCurr1';
	tyMpNtParamMpLink : MpComIdentType;
END_VAR
(**)
(*Local*)
VAR
	bRstErr : BOOL;
	udiRstErrOld : UDINT;
	bInitDone : BOOL;
	bInitialDone : BOOL;
	usiStep : USINT;
	fbMpNtParamRegPar : MpRecipeRegPar;
	fbMpNtParamXml : MpRecipeXml;
	fbDirCreate1 : fbDirCreate;
	fbDirCreate2 : fbDirCreate;
	fbDirCreate3 : fbDirCreate;
	fbFileRead1 : fbFileFullReadEncry;
	fbFileWrite1 : fbFileFullWriteEncry;
	udiModuleNum : UDINT := 5151;
END_VAR
```

#### Act_Action.st
```iecst
(** 2019-03-25 **)
ACTION Act_Action:

	//Reset Error
	IF (eStatus = Error) AND bRstErr THEN
		p_eAct	:= NtParamActIdle;
		eStat	:= NtParamActIdle;
	END_IF

	//Reset Done
	IF eStatus = Done AND p_eAct = NtParamActIdle THEN
		eStat	:= NtParamActIdle;
	END_IF

	//Set p_eAct
	IF eStatus = Idle THEN
		eStat	:= p_eAct;
	END_IF

END_ACTION
```

#### Act_Alarm.st
```iecst
(** 2019-03-25 **)
ACTION Act_Alarm:

	//Error
	IF EDGEPOS(eStatus = Error) THEN

		tyAlmData.sProgNm		:= p_sProgNm;
		tyAlmData.udiCode		:= udiStatus;
		tyAlmData.eSeverity		:= AlmSeverityError;
		tyAlmData.udiRunTime	:= tyAlmData.udiRunTime + 1;
		tyAlmData.bAlm			:= TRUE;
		tyAlmData.udiModuleNum  := udiModuleNum;
		g_sNtParamProgNm		:= p_sProgNm;

		//Get Error Message
		IF tyAlmData.udiCode < 10000 OR tyAlmData.udiCode > 10099 THEN
			tyAlmData.sAlmMsg	:= 'Unknown';
			tyAlmData.sRcyMsg	:= 'Unknown';
		ELSE
			tyAlmData.sAlmMsg	:= a_tyAlmText[tyAlmData.udiCode].sAlmText;
			tyAlmData.sRcyMsg	:= a_tyAlmText[tyAlmData.udiCode].sRcyText;
		END_IF

		sStatTxt	:= tyAlmData.sAlmMsg;

	ELSIF bRstErr AND (tyAlmData.udiCode <> 0) THEN

		tyAlmData.udiCode	:= 0;
		tyAlmData.eSeverity	:= AlmSeverityNA;
		tyAlmData.sAlmMsg	:= '';
		tyAlmData.sRcyMsg	:= '';
		tyAlmData.bAlm			:= FALSE;
		sStatTxt	:= a_sStatText[eStat];

	END_IF

END_ACTION
```

#### Act_InitGlobal.st
```iecst
(** 2019-03-25 **)
ACTION Act_InitGlobal:

	(* Always Change If Project Change *)

	//Pass Data To Link
	p_bLinkStartupRun ACCESS p_StartupRun;

	//Pass Data To Internal Use
	p_udiRstErr ACCESS p_RstErrReset;

	(* Always Change If Project Change *)

END_ACTION
```

#### Act_Initial.st
```iecst
(** 2020-07-27 **)
ACTION Act_Initial:

	//Initial
	sStatTxt	:= a_sStatText[eStat];

	fbDirCreate1.sDevice	:= 'F';
	fbDirCreate1.sDirName	:= 'Private';
	fbDirCreate1(bEn := FALSE);

	fbDirCreate2.sDevice	:= 'Private';
	fbDirCreate2.sDirName	:= 'NutekParameter';
	fbDirCreate2(bEn := FALSE);

	fbDirCreate3.sDevice	:= 'Private';
	fbDirCreate3.sDirName	:= 'NutekParameterXml';
	fbDirCreate3(bEn := FALSE);

	fbFileRead1.sDevice			:= 'NtParam';
	fbFileRead1.sFile			:= p_sFileName;
	fbFileRead1.udiOffset		:= 0;
	fbFileRead1.p_Dest			:= ADR(tyNtParamCurr);
	fbFileRead1.udiLen			:= SIZEOF(tyNtParamCurr);
	fbFileRead1.usiEncryptCode	:= 130;
	fbFileRead1(bEn := FALSE);

	fbFileWrite1.sDevice		:= 'NtParam';
	fbFileWrite1.sFile			:= p_sFileName;
	fbFileWrite1.udiOffset		:= 0;
	fbFileWrite1.p_Src			:= ADR(tyNtParamCurr);
	fbFileWrite1.udiLen			:= SIZEOF(tyNtParamCurr);
	fbFileWrite1.udiOption		:= 0;
	fbFileWrite1.usiEncryptCode	:= 130;
	fbFileWrite1(bEn := FALSE);

	tyMpNtParamMpLink	:= gRecipeXml;

	fbMpNtParamRegPar.MpLink	:= ADR(tyMpNtParamMpLink);
	fbMpNtParamRegPar.PVName	:= ADR(p_sPVName);
	fbMpNtParamRegPar(Enable := FALSE);

	fbMpNtParamXml.MpLink		:= ADR(tyMpNtParamMpLink);
	fbMpNtParamXml.DeviceName	:= ADR('MpNtParam');
	fbMpNtParamXml.FileName		:= ADR(p_sFileName1);
	fbMpNtParamXml(Enable := FALSE);

END_ACTION
```

#### Act_InitLocal.st
```iecst
(** 2020-07-27 **)
ACTION Act_InitLocal:

	//Input Reference Link To Local Variable
	p_eAct ACCESS ADR(eAct);
	p_udiRstErr ACCESS ADR(udiRstErr);
	p_sFileName ACCESS ADR(sFileName);
	p_sProgNm ACCESS ADR(sProgNm);
	p_tyMpNtParamMpLink ACCESS ADR(tyMpNtParamMpLink);
	p_sFileName1 ACCESS ADR(sFileName1);
	p_sPVName ACCESS ADR(sPVName);

END_ACTION
```

#### Act_LinkAction.st
```iecst
(** 2019-04-09 **)
ACTION Act_LinkAction:

	IF p_bLinkStartupRun = TRUE THEN
		p_eAct ACCESS p_StartupNtParamAct;
	ELSE
		p_eAct ACCESS ADR(eAct);
	END_IF

END_ACTION
```

#### Act_Main.st
```iecst
(** 2020-07-27 **)
ACTION Act_Main:

	//Main
	CASE eStat OF

		NtParamActIdle:
			IF eStatus <> Idle THEN	//Reset Data
				//Private
				fbDirCreate1(bEn := FALSE);
				fbDirCreate2(bEn := FALSE);
				fbDirCreate3(bEn := FALSE);
				fbFileRead1(bEn := FALSE);
				fbFileWrite1(bEn := FALSE);
				fbMpNtParamRegPar(Enable := FALSE);
				fbMpNtParamXml(Enable := FALSE);
				usiStep	:= 0;

				bFileNotFound	:= FALSE;

				sStatTxt	:= a_sStatText[eStat];

			END_IF

			eStatus	:= Idle;

		NtParamActCreateDir:
			IF eStatus = Idle OR eStatus = Busy THEN

				eStatus	:= Busy;

				sStatTxt	:= a_sStatText[eStat];

				CASE usiStep OF
					0:
						fbDirCreate1(bEn := TRUE);
						IF fbDirCreate1.udiStatus = 0 THEN
							usiStep	:= 1;
						ELSIF fbDirCreate1.udiStatus < 65534 THEN
							eStatus		:= Error;

							IF fbDirCreate1.udiStatus = 1908 THEN
								udiStatus	:= 10000;	//Create User Directory Error
							ELSE
								udiStatus	:= fbDirCreate1.udiStatus;
							END_IF
						END_IF

					1:
						fbDirCreate2(bEn := TRUE);
						IF fbDirCreate2.udiStatus = 0 THEN
							usiStep	:= 2;
						ELSIF fbDirCreate2.udiStatus < 65534 THEN
							eStatus		:= Error;

							IF fbDirCreate2.udiStatus = 1908 THEN
								udiStatus	:= 10001;	//Create Nutek Parameter Directory Error
							ELSE
								udiStatus	:= fbDirCreate2.udiStatus;
							END_IF
						END_IF

					2:
						fbDirCreate3(bEn := TRUE);
						IF fbDirCreate3.udiStatus = 0 THEN
							eStatus	:= Done;
						ELSIF fbDirCreate3.udiStatus < 65534 THEN
							eStatus		:= Error;

							IF fbDirCreate3.udiStatus = 1908 THEN
								udiStatus	:= 10014;	//Create Nutek Parameter xml Directory Error
							ELSE
								udiStatus	:= fbDirCreate3.udiStatus;
							END_IF
						END_IF

				END_CASE

			END_IF

		NtParamActWrite:
			IF eStatus = Idle OR eStatus = Busy THEN

				eStatus	:= Busy;

				sStatTxt	:= a_sStatText[eStat];

				fbFileWrite1(bEn := TRUE);
				IF fbFileWrite1.udiStatus = 0 THEN
					eStatus			:= Done;
				ELSIF fbFileWrite1.udiStatus < 65534 THEN
					eStatus			:= Error;

					IF fbFileWrite1.udiStatus = 1900 THEN
						udiStatus	:= 10002;	//File Open Error While Writing
					ELSIF fbFileWrite1.udiStatus = 1901 THEN
						udiStatus	:= 10003;	//File Create Error While Writing
					ELSIF fbFileWrite1.udiStatus = 1903 THEN
						udiStatus	:= 10004;	//File Write Error
					ELSIF fbFileWrite1.udiStatus = 1904 THEN
						udiStatus	:= 10005;	//File Close Error While Writing
					ELSIF fbFileWrite1.udiStatus = 1914 THEN
						udiStatus	:= 10009;	//Directory Does Not Exist While Writing
					ELSE
						udiStatus	:= fbFileWrite1.udiStatus;
					END_IF
				END_IF

			END_IF

		NtParamActRead:
			IF eStatus = Idle OR eStatus = Busy THEN

				eStatus	:= Busy;

				sStatTxt	:= a_sStatText[eStat];

				fbFileRead1(bEn := TRUE);
				IF fbFileRead1.udiStatus = 0 THEN
					eStatus			:= Done;
				ELSIF fbFileRead1.udiStatus < 65534 THEN
					eStatus		:= Error;

					IF fbFileRead1.udiStatus = 1900 THEN
						udiStatus	:= 10006;	//File Open Error While Reading
					ELSIF fbFileRead1.udiStatus = 1902 THEN
						udiStatus	:= 10007;	//File Read Error
					ELSIF fbFileRead1.udiStatus = 1904 THEN
						udiStatus	:= 10008;	//File Close Error While Reading
					ELSIF fbFileRead1.udiStatus = 1915 THEN
						eStatus			:= Done;
						bFileNotFound	:= TRUE;
					ELSE
						udiStatus	:= fbFileRead1.udiStatus;
					END_IF
				END_IF

			END_IF

		NtParamActLoad:
			IF eStatus = Idle OR eStatus = Busy THEN

				eStatus	:= Busy;

				sStatTxt	:= a_sStatText[eStat];

				CASE usiStep OF
					0:
						fbMpNtParamRegPar(Enable := TRUE);

						IF (fbMpNtParamRegPar.Active = TRUE) AND (fbMpNtParamRegPar.StatusID = 0) THEN
							usiStep	:= 1;
						ELSIF fbMpNtParamRegPar.StatusID <> 0 THEN
							eStatus		:= Error;
							udiStatus	:= 10010;	//MpRecipeRegPar Error While Loading
						END_IF

					1:
						fbMpNtParamXml.Load	:= TRUE;
						fbMpNtParamXml.Save	:= FALSE;
						fbMpNtParamXml(Enable := TRUE);

						IF (fbMpNtParamXml.Active = TRUE) AND (fbMpNtParamXml.CommandDone = TRUE) AND (fbMpNtParamXml.StatusID = 0) THEN
							//	eStatus	:= Done;
							usiStep	:= 2;
							tyNtParamCurr	:= tyMpNtParamCurr1;
						ELSIF fbMpNtParamXml.StatusID <> 0 THEN
							eStatus		:= Error;
							udiStatus	:= 10011;	//MpRecipeXml Error While Loading
						END_IF

					2:
						fbFileWrite1(bEn := TRUE);
						IF fbFileWrite1.udiStatus = 0 THEN
							eStatus			:= Done;
						ELSIF fbFileWrite1.udiStatus < 65534 THEN
							eStatus			:= Error;

							IF fbFileWrite1.udiStatus = 1900 THEN
								udiStatus	:= 10002;	//File Open Error While Writing
							ELSIF fbFileWrite1.udiStatus = 1901 THEN
								udiStatus	:= 10003;	//File Create Error While Writing
							ELSIF fbFileWrite1.udiStatus = 1903 THEN
								udiStatus	:= 10004;	//File Write Error
							ELSIF fbFileWrite1.udiStatus = 1904 THEN
								udiStatus	:= 10005;	//File Close Error While Writing
							ELSIF fbFileWrite1.udiStatus = 1914 THEN
								udiStatus	:= 10009;	//Directory Does Not Exist While Writing
							ELSE
								udiStatus	:= fbFileWrite1.udiStatus;
							END_IF
						END_IF

				END_CASE

			END_IF

		NtParamActSave:
			IF eStatus = Idle OR eStatus = Busy THEN

				eStatus	:= Busy;

				sStatTxt	:= a_sStatText[eStat];

				CASE usiStep OF
					0:
						tyMpNtParamCurr1	:= tyNtParamCurr;
						fbMpNtParamRegPar(Enable := TRUE);

						IF (fbMpNtParamRegPar.Active = TRUE) AND (fbMpNtParamRegPar.StatusID = 0) THEN
							usiStep	:= 1;
						ELSIF fbMpNtParamRegPar.StatusID <> 0 THEN
							eStatus		:= Error;
							udiStatus	:= 10012;	//MpRecipeRegPar Error While Saving
						END_IF

					1:
						fbMpNtParamXml.Load	:= FALSE;
						fbMpNtParamXml.Save	:= TRUE;
						fbMpNtParamXml(Enable := TRUE);

						IF (fbMpNtParamXml.Active = TRUE) AND (fbMpNtParamXml.CommandDone = TRUE) AND (fbMpNtParamXml.StatusID = 0) THEN
							eStatus	:= Done;
						ELSIF fbMpNtParamXml.StatusID <> 0 THEN
							eStatus		:= Error;
							udiStatus	:= 10013;	//MpRecipeXml Error While Saving
						END_IF

				END_CASE

			END_IF

	END_CASE

END_ACTION
```

#### Cyclic.st
```iecst
(** 2019-03-29 **)
PROGRAM _CYCLIC

	IF bInitDone = FALSE THEN
		bInitDone	:= TRUE;

		Act_InitLocal;
		Act_InitGlobal;

	ELSIF bInitialDone = FALSE THEN
		bInitialDone	:= TRUE;

		Act_Initial;

	ELSE

		Act_RstErr;
		Act_LinkAction;
		Act_Action;
		Act_Link;
		Act_Main;
		Act_Alarm;

	END_IF

END_PROGRAM
```

#### Init.st
```iecst
(** 2020-10-06 **)
PROGRAM _INIT

	(* Always Change If Project Change *)

	//Pass Address To Global Address For External Use
	//Action, State & Status
	p_NtParamStat		:= ADR(eStat);
	p_NtParamStatus		:= ADR(eStatus);
	p_NtParamStatTxt	:= ADR(sStatTxt);

	//Alarm
	p_NtParamAlmData	:= ADR(tyAlmData);

	//Output
	p_NtParamFileNotFound			:= ADR(bFileNotFound);

	p_NtParamCurr					:= ADR(tyNtParamCurr);
	p_NtParamDISettings				:= ADR(tyNtParamCurr.tyDISettings);
	p_NtParamDOSettings				:= ADR(tyNtParamCurr.tyDOSettings);
	p_NtParamAWPrep					:= ADR(tyNtParamCurr.bAWPrep);
	p_NtParamLFPrep					:= ADR(tyNtParamCurr.bLFPrep);
	p_NtParamLeaderMc				:= ADR(tyNtParamCurr.bLeaderMc);
	p_NtParamLFUsrSetPrep			:= ADR(tyNtParamCurr.bLFUsrSetPrep);
	p_NtParamLFWidthLimit			:= ADR(tyNtParamCurr.diLFWidthLimit);
	p_NtParamLFProdWidthChk			:= ADR(tyNtParamCurr.bLFProdWidthChk);
	p_NtParamUSWidthChkPrep			:= ADR(tyNtParamCurr.bUSWidthChkPrep);
	p_NtParamDSWidthChkPrep			:= ADR(tyNtParamCurr.bDSWidthChkPrep);
	p_NtParamLCSLFPrep				:= ADR(tyNtParamCurr.bLCSLFPrep);
	p_NtParamLCSReqRcpPrep			:= ADR(tyNtParamCurr.bLCSReqRcpPrep);
	p_NtParamLCSManageRcpPrep		:= ADR(tyNtParamCurr.bLCSManageRcpPrep);
	p_NtParamLCSLiveDatPrep			:= ADR(tyNtParamCurr.bLCSLiveDatPrep);
	p_NtParamUSExtSMEMAPrep			:= ADR(tyNtParamCurr.bUSExtSMEMAPrep);
	p_NtParamDSExtSMEMAPrep			:= ADR(tyNtParamCurr.bDSExtSMEMAPrep);
	p_NtParamVSMEMAPrep				:= ADR(tyNtParamCurr.bVSMEMAPrep);
	p_NtParamHermesPrep				:= ADR(tyNtParamCurr.bHermesPrep);
	p_NtParamHermesRmtPrep			:= ADR(tyNtParamCurr.bHermesRmtPrep);
	p_NtParamSSaverPrep				:= ADR(tyNtParamCurr.bSSaverPrep);
	p_NtParamWidthOffset			:= ADR(tyNtParamCurr.diWidthOffsetInUM);
	p_NtParamJobNo					:= ADR(tyNtParamCurr.sJobNo);
	p_NtParamNtAddr					:= ADR(tyNtParamCurr.usiNtAddr);

	p_NtParamProjConvDir			:= ADR(tyNtParamCurr.eProjConvDir);
	p_NtParamProjBypsInitConvPrep	:= ADR(tyNtParamCurr.bProjBypsInitConvPrep);
	p_NtParamProjCoatingPrep		:= ADR(tyNtParamCurr.bProjCoatingPrep);
	p_NtParamProjStopperPrep		:= ADR(tyNtParamCurr.bProjStopperPrep);
	p_NtParamProjClampPrep			:= ADR(tyNtParamCurr.bProjClampPrep);
	p_NtParamProjClampOption		:= ADR(tyNtParamCurr.eProjClampOption);
	p_NtParamProjInletShutPrep		:= ADR(tyNtParamCurr.bProjInletShutPrep);
	p_NtParamProjOutletShutPrep		:= ADR(tyNtParamCurr.bProjOutletShutPrep);
	p_NtParamProjRlsNewProdPrep		:= ADR(tyNtParamCurr.bProjRlsNewProdPrep);

	p_NtParamUsrFolderProgNm		:= ADR(tyNtParamCurr.sUsrFolderProgNm);

	p_NtParamLibVersionProgNm		:= ADR(tyNtParamCurr.sLibVersionProgNm);

	p_NtParamTimeProgNm				:= ADR(tyNtParamCurr.sTimeProgNm);

	p_NtParamHWInfoProgNm			:= ADR(tyNtParamCurr.sHWInfoProgNm);
	p_NtParamHWInfoDevice			:= ADR(tyNtParamCurr.sHWInfoDevice);

	p_NtParamTLChgRcpBlinkTm		:= ADR(tyNtParamCurr.tTLChgRcpBlinkTm);

	p_NtParamTLErrBlinkTm			:= ADR(tyNtParamCurr.tTLErrBlinkTm);
	p_NtParamBuzErrOnTm				:= ADR(tyNtParamCurr.tBuzErrOnTm);
	p_NtParamBuzErrRestTm			:= ADR(tyNtParamCurr.tBuzErrRestTm);
	p_NtParamBuzErrOnCntr			:= ADR(tyNtParamCurr.usiBuzErrOnCntr);
	p_NtParamBuzErrStopSeqEn		:= ADR(tyNtParamCurr.bBuzErrStopSeqEn);
	p_NtParamBuzErrStopSeqCntr		:= ADR(tyNtParamCurr.usiBuzErrStopSeqCntr);

	p_NtParamTLWarnBlinkTm			:= ADR(tyNtParamCurr.tTLWarnBlinkTm);
	p_NtParamBuzWarnOnTm			:= ADR(tyNtParamCurr.tBuzWarnOnTm);
	p_NtParamBuzWarnRestTm			:= ADR(tyNtParamCurr.tBuzWarnRestTm);
	p_NtParamBuzWarnOnCntr			:= ADR(tyNtParamCurr.usiBuzWarnOnCntr);
	p_NtParamBuzWarnStopSeqEn		:= ADR(tyNtParamCurr.bBuzWarnStopSeqEn);
	p_NtParamBuzWarnStopSeqCntr		:= ADR(tyNtParamCurr.usiBuzWarnStopSeqCntr);

	p_NtParamTLWarn1BlinkTm			:= ADR(tyNtParamCurr.tTLWarn1BlinkTm);
	p_NtParamBuzWarn1OnTm			:= ADR(tyNtParamCurr.tBuzWarn1OnTm);
	p_NtParamBuzWarn1RestTm			:= ADR(tyNtParamCurr.tBuzWarn1RestTm);
	p_NtParamBuzWarn1OnCntr			:= ADR(tyNtParamCurr.usiBuzWarn1OnCntr);
	p_NtParamBuzWarn1StopSeqEn		:= ADR(tyNtParamCurr.bBuzWarn1StopSeqEn);
	p_NtParamBuzWarn1StopSeqCntr	:= ADR(tyNtParamCurr.usiBuzWarn1StopSeqCntr);

	p_NtParamTLWarn2BlinkTm			:= ADR(tyNtParamCurr.tTLWarn2BlinkTm);
	p_NtParamBuzWarn2OnTm			:= ADR(tyNtParamCurr.tBuzWarn2OnTm);
	p_NtParamBuzWarn2RestTm			:= ADR(tyNtParamCurr.tBuzWarn2RestTm);
	p_NtParamBuzWarn2OnCntr			:= ADR(tyNtParamCurr.usiBuzWarn2OnCntr);
	p_NtParamBuzWarn2StopSeqEn		:= ADR(tyNtParamCurr.bBuzWarn2StopSeqEn);
	p_NtParamBuzWarn2StopSeqCntr	:= ADR(tyNtParamCurr.usiBuzWarn2StopSeqCntr);

	p_NtParamTLWarn3BlinkTm			:= ADR(tyNtParamCurr.tTLWarn3BlinkTm);
	p_NtParamBuzWarn3OnTm			:= ADR(tyNtParamCurr.tBuzWarn3OnTm);
	p_NtParamBuzWarn3RestTm			:= ADR(tyNtParamCurr.tBuzWarn3RestTm);
	p_NtParamBuzWarn3OnCntr			:= ADR(tyNtParamCurr.usiBuzWarn3OnCntr);
	p_NtParamBuzWarn3StopSeqEn		:= ADR(tyNtParamCurr.bBuzWarn3StopSeqEn);
	p_NtParamBuzWarn3StopSeqCntr	:= ADR(tyNtParamCurr.usiBuzWarn3StopSeqCntr);

	p_NtParamTLWarn4BlinkTm			:= ADR(tyNtParamCurr.tTLWarn4BlinkTm);
	p_NtParamBuzWarn4OnTm			:= ADR(tyNtParamCurr.tBuzWarn4OnTm);
	p_NtParamBuzWarn4RestTm			:= ADR(tyNtParamCurr.tBuzWarn4RestTm);
	p_NtParamBuzWarn4OnCntr			:= ADR(tyNtParamCurr.usiBuzWarn4OnCntr);
	p_NtParamBuzWarn4StopSeqEn		:= ADR(tyNtParamCurr.bBuzWarn4StopSeqEn);
	p_NtParamBuzWarn4StopSeqCntr	:= ADR(tyNtParamCurr.usiBuzWarn4StopSeqCntr);

	p_NtParamTLWarn5BlinkTm			:= ADR(tyNtParamCurr.tTLWarn5BlinkTm);
	p_NtParamBuzWarn5OnTm			:= ADR(tyNtParamCurr.tBuzWarn5OnTm);
	p_NtParamBuzWarn5RestTm			:= ADR(tyNtParamCurr.tBuzWarn5RestTm);
	p_NtParamBuzWarn5OnCntr			:= ADR(tyNtParamCurr.usiBuzWarn5OnCntr);
	p_NtParamBuzWarn5StopSeqEn		:= ADR(tyNtParamCurr.bBuzWarn5StopSeqEn);
	p_NtParamBuzWarn5StopSeqCntr	:= ADR(tyNtParamCurr.usiBuzWarn5StopSeqCntr);

	p_NtParamBuzAlertOnTm			:= ADR(tyNtParamCurr.tBuzAlertOnTm);
	p_NtParamBuzAlertRestTm			:= ADR(tyNtParamCurr.tBuzAlertRestTm);
	p_NtParamBuzAlertOnCntr			:= ADR(tyNtParamCurr.usiBuzAlertOnCntr);
	p_NtParamBuzAlertStopSeqEn		:= ADR(tyNtParamCurr.bBuzAlertStopSeqEn);
	p_NtParamBuzAlertStopSeqCntr	:= ADR(tyNtParamCurr.usiBuzAlertStopSeqCntr);

	p_NtParamTLBlueBlinkTm			:= ADR(tyNtParamCurr.tTLBlueBlinkTm);
	p_NtParamTLAmberBlinkTm			:= ADR(tyNtParamCurr.tTLAmberBlinkTm);
	p_NtParamTLWhiteBlinkTm			:= ADR(tyNtParamCurr.tTLWhiteBlinkTm);
	p_NtParamTLRedBlinkTm			:= ADR(tyNtParamCurr.tTLRedBlinkTm);
	p_NtParamTLGreenBlinkTm			:= ADR(tyNtParamCurr.tTLGreenBlinkTm);

	p_NtParamTLBuzMode				:= ADR(tyNtParamCurr.eTLBuzMode);

	p_NtParamAlmProgNm				:= ADR(tyNtParamCurr.sAlmProgNm);
	p_NtParamAlmFileKeepDay			:= ADR(tyNtParamCurr.udiAlmFileKeepDay);

	p_NtParamProdRcpProgNm			:= ADR(tyNtParamCurr.sProdRcpProgNm);
	p_NtParamProdRcpListFileNm		:= ADR(tyNtParamCurr.sProdRcpListFileNm);
	p_NtParamProdRcpSingleFileNm	:= ADR(tyNtParamCurr.sProdRcpSingleFileNm);

	p_NtParamMpProdRcpProgNm		:= ADR(tyNtParamCurr.sMpProdRcpProgNm);
	p_NtParamMpProdRcpFileNm		:= ADR(tyNtParamCurr.sMpProdRcpFileNm);
	p_NtParamMpProdRcpPVNm			:= ADR(tyNtParamCurr.sMpProdRcpPVNm);

	p_NtParamMcParamProgNm			:= ADR(tyNtParamCurr.sMcParamProgNm);
	p_NtParamMcParamFileNm			:= ADR(tyNtParamCurr.sMcParamFileNm);

	p_NtParamUsrMgmtProgNm			:= ADR(tyNtParamCurr.sUsrMgmtProgNm);

	p_NtParamUSSMEMAProgNm			:= ADR(tyNtParamCurr.sUSSMEMAProgNm);
	p_NtParamUSSMEMARstDlyTm		:= ADR(tyNtParamCurr.tUSSMEMARstDlyTm);
	p_NtParamUSSMEMASigInChkTm		:= ADR(tyNtParamCurr.tUSSMEMASigInChkTm);

	p_NtParamDSSMEMAProgNm			:= ADR(tyNtParamCurr.sDSSMEMAProgNm);
	p_NtParamDSSMEMARstDlyTm		:= ADR(tyNtParamCurr.tDSSMEMARstDlyTm);
	p_NtParamDSSMEMASigInChkTm		:= ADR(tyNtParamCurr.tDSSMEMASigInChkTm);

	p_NtParamConvProgNm				:= ADR(tyNtParamCurr.sConvProgNm);
	p_NtParamConvOnDirMod			:= ADR(tyNtParamCurr.bConvOnDirMod);
	p_NtParamConvMtrOffDlyTm		:= ADR(tyNtParamCurr.tConvMtrOffDlyTm);
	p_NtParamConvFwdDlyTm			:= ADR(tyNtParamCurr.diConvFwdDlyTm);
	p_NtParamConvRevDlyTm			:= ADR(tyNtParamCurr.diConvRevDlyTm);

	p_NtParamStopperProgNm			:= ADR(tyNtParamCurr.sStopperProgNm);
	p_NtParamStopperTwoCtrlIn		:= ADR(tyNtParamCurr.bStopperTwoCtrlIn);
	p_NtParamStopperExtDlyTm		:= ADR(tyNtParamCurr.tStopperExtDlyTm);
	p_NtParamStopperRetDlyTm		:= ADR(tyNtParamCurr.tStopperRetDlyTm);

	p_NtParamClampProgNm			:= ADR(tyNtParamCurr.sClampProgNm);
	p_NtParamClampTwoCtrlIn			:= ADR(tyNtParamCurr.bClampTwoCtrlIn);
	p_NtParamClampExtDlyTm			:= ADR(tyNtParamCurr.tClampExtDlyTm);
	p_NtParamClampRetDlyTm			:= ADR(tyNtParamCurr.tClampRetDlyTm);

	p_NtParamInShutterProgNm		:= ADR(tyNtParamCurr.sInShutterProgNm);
	p_NtParamInShutterTwoCtrlIn		:= ADR(tyNtParamCurr.bInShutterTwoCtrlIn);
	p_NtParamInShutterExtTO			:= ADR(tyNtParamCurr.tInShutterExtTO);
	p_NtParamInShutterRetTO			:= ADR(tyNtParamCurr.tInShutterRetTO);

	p_NtParamOutShutterProgNm		:= ADR(tyNtParamCurr.sOutShutterProgNm);
	p_NtParamOutShutterTwoCtrlIn	:= ADR(tyNtParamCurr.bOutShutterTwoCtrlIn);
	p_NtParamOutShutterExtTO		:= ADR(tyNtParamCurr.tOutShutterExtTO);
	p_NtParamOutShutterRetTO		:= ADR(tyNtParamCurr.tOutShutterRetTO);

	p_NtParamClamp1ProgNm			:= ADR(tyNtParamCurr.sClamp1ProgNm);
	p_NtParamClamp1TwoCtrlIn		:= ADR(tyNtParamCurr.bClamp1TwoCtrlIn);
	p_NtParamClamp1ExtTO			:= ADR(tyNtParamCurr.tClamp1ExtTO);
	p_NtParamClamp1RetTO			:= ADR(tyNtParamCurr.tClamp1RetTO);

	p_NtParamClamp2ProgNm			:= ADR(tyNtParamCurr.sClamp2ProgNm);
	p_NtParamClamp2TwoCtrlIn		:= ADR(tyNtParamCurr.bClamp2TwoCtrlIn);
	p_NtParamClamp2ExtTO			:= ADR(tyNtParamCurr.tClamp2ExtTO);
	p_NtParamClamp2RetTO			:= ADR(tyNtParamCurr.tClamp2RetTO);

	p_NtParamClamp3ProgNm			:= ADR(tyNtParamCurr.sClamp3ProgNm);
	p_NtParamClamp3TwoCtrlIn		:= ADR(tyNtParamCurr.bClamp3TwoCtrlIn);
	p_NtParamClamp3ExtTO			:= ADR(tyNtParamCurr.tClamp3ExtTO);
	p_NtParamClamp3RetTO			:= ADR(tyNtParamCurr.tClamp3RetTO);

	p_NtParamMotorOnDlyTm			:= ADR(tyNtParamCurr.diMotorOnDlyTm);
	p_NtParamMotorOffDlyTm			:= ADR(tyNtParamCurr.diMotorOffDlyTm);
	p_NtParamBrakeOnDlyTm			:= ADR(tyNtParamCurr.diBrakeOnDlyTm);
	p_NtParamBrakeOffDlyTm			:= ADR(tyNtParamCurr.diBrakeOffDlyTm);
	p_NtParamTimeOut				:= ADR(tyNtParamCurr.diTimeOut);

	p_NtParamAWProgNm				:= ADR(tyNtParamCurr.sAWProgNm);
	p_NtParamAWDevice				:= ADR(tyNtParamCurr.sAWDevice);
	p_NtParamAWNode					:= ADR(tyNtParamCurr.usiAWNode);
	p_NtParamAWDir					:= ADR(tyNtParamCurr.bAWDir);
	p_NtParamAWDirBl				:= ADR(tyNtParamCurr.bAWDirBl);
	p_NtParamAWPitchInUM			:= ADR(tyNtParamCurr.diAWPitchInUM);
	p_NtParamAWMovBlDistInUM		:= ADR(tyNtParamCurr.diAWMovBlDistInUM);
	p_NtParamAWParamInHm			:= ADR(tyNtParamCurr.tyAWParamInHm);
	p_NtParamAWParamInConvert		:= ADR(tyNtParamCurr.tyAWParamInConvert);
	p_NtParamAWParam				:= ADR(tyNtParamCurr.tyAWParam);
	p_NtParamAWAcc					:= ADR(tyNtParamCurr.tyAWParam.diAccInMS);
	p_NtParamAWDec					:= ADR(tyNtParamCurr.tyAWParam.diDecInMS);
	p_NtParamAWAutoSpd				:= ADR(tyNtParamCurr.tyAWParam.diAutoSpdInUMPS);
	p_NtParamAWTuning				:= ADR(tyNtParamCurr.tyAWTuning);
	p_NtParamAWMotorType			:= ADR(tyNtParamCurr.eAWServoMotorType);

	p_NtParamInvertProgNm			:= ADR(tyNtParamCurr.sInvertProgNm);
	p_NtParamInvertDevice			:= ADR(tyNtParamCurr.sInvertDevice);
	p_NtParamInvertNode				:= ADR(tyNtParamCurr.usiInvertNode);
	p_NtParamInvertDir				:= ADR(tyNtParamCurr.bInvertDir);
	p_NtParamInvertParamInHm		:= ADR(tyNtParamCurr.tyInvertParamInHm);
	p_NtParamInvertParamInConvert	:= ADR(tyNtParamCurr.tyInvertParamInConvert);
	p_NtParamInvertParam			:= ADR(tyNtParamCurr.tyInvertParam);
	p_NtParamInvertAcc				:= ADR(tyNtParamCurr.tyInvertParam.diAccInMS);
	p_NtParamInvertDec				:= ADR(tyNtParamCurr.tyInvertParam.diDecInMS);
	p_NtParamInvertAutoSpd			:= ADR(tyNtParamCurr.tyInvertParam.diAutoSpdInUMPS);
	p_NtParamInvertTuning			:= ADR(tyNtParamCurr.tyInvertTuning);
	p_NtParamInvertMotorType		:= ADR(tyNtParamCurr.eInvertServoMotorType);

	p_NtParamDInputProgNm			:= ADR(tyNtParamCurr.sDIProgNm);

	p_NtParamMcProgNm				:= ADR(tyNtParamCurr.sMcProgNm);

	p_NtParamHermesProgNm			:= ADR(tyNtParamCurr.sHermesProgNm);
	p_NtParamHermesRetainFileNm		:= ADR(tyNtParamCurr.sHermesRetainFileNm);
	p_NtParamHermesConfigFileNm		:= ADR(tyNtParamCurr.sHermesConfigFileNm);

	p_NtParamUSHermesProgNm			:= ADR(tyNtParamCurr.sUSHermesProgNm);
	p_NtParamUSHermesFileKeepDay	:= ADR(tyNtParamCurr.udiUSHermesFileKeepDay);
	p_NtParamUSHermesAliveTmInSec	:= ADR(tyNtParamCurr.udiUSHermesAliveTmInSec);
	p_NtParamUSHermesConnTO			:= ADR(tyNtParamCurr.tUSHermesConnTO);
	//US Hermes 2
	p_NtParamUSHermes2ProgNm			:= ADR(tyNtParamCurr.sUSHermes2ProgNm);
	p_NtParamUSHermes2FileKeepDay		:= ADR(tyNtParamCurr.udiUSHermes2FileKeepDay);
	p_NtParamUSHermes2AliveTmInSec		:= ADR(tyNtParamCurr.udiUSHermes2AliveTmInSec);
	p_NtParamUSHermes2ConnTO			:= ADR(tyNtParamCurr.tUSHermes2ConnTO);

	p_NtParamDSHermesProgNm			:= ADR(tyNtParamCurr.sDSHermesProgNm);
	p_NtParamDSHermesFileKeepDay	:= ADR(tyNtParamCurr.udiDSHermesFileKeepDay);
	p_NtParamDSHermesAliveTmInSec	:= ADR(tyNtParamCurr.udiDSHermesAliveTmInSec);
	p_NtParamDSHermesConnTO			:= ADR(tyNtParamCurr.tDSHermesConnTO);
	//DS Hermes2
	p_NtParamDSHermes2ProgNm		:= ADR(tyNtParamCurr.sDSHermesProgNm);
	p_NtParamDSHermes2FileKeepDay	:= ADR(tyNtParamCurr.udiDSHermesFileKeepDay);
	p_NtParamDSHermes2AliveTmInSec	:= ADR(tyNtParamCurr.udiDSHermesAliveTmInSec);
	p_NtParamDSHermes2ConnTO		:= ADR(tyNtParamCurr.tDSHermesConnTO);

	p_NtParamRmtHermesProgNm		:= ADR(tyNtParamCurr.sRmtHermesProgNm);
	p_NtParamRmtHermesConfigFileNm	:= ADR(tyNtParamCurr.sRmtHermesConfigFileNm);
	p_NtParamRmtHermesFileKeepDay	:= ADR(tyNtParamCurr.udiRmtHermesFileKeepDay);
	p_NtParamRmtHermesAliveTmInSec	:= ADR(tyNtParamCurr.udiRmtHermesAliveTmInSec);
	p_NtParamRmtHermesSndBffrSize	:= ADR(tyNtParamCurr.udiRmtHermesSndBffrSize);
	p_NtParamRmtHermesRcvBffrSize	:= ADR(tyNtParamCurr.udiRmtHermesRcvBffrSize);

	p_NtParamOpsAWProgNm			:= ADR(tyNtParamCurr.sOpsAWProgNm);
	p_NtParamOpsInitConvProgNm		:= ADR(tyNtParamCurr.sOpsInitConvProgNm);
	p_NtParamOpsInitPneuProgNm		:= ADR(tyNtParamCurr.sOpsInitPneuProgNm);
	p_NtParamOpsConvProgNm			:= ADR(tyNtParamCurr.sOpsConvProgNm);
	p_NtParamOpsPneuProgNm			:= ADR(tyNtParamCurr.sOpsPneuProgNm);

	p_NtParamConvBffrProgNm			:= ADR(tyNtParamCurr.sConvBffrProgNm);
	p_NtParamConvBffrFileNm			:= ADR(tyNtParamCurr.sConvBffrFileNm);
	p_NtParamConvBffrIdx			:= ADR(tyNtParamCurr.iConvBffrIdx);

	p_NtParamLFLeaderProgNm			:= ADR(tyNtParamCurr.sLFLeaderProgNm);
	p_NtParamLFLeaderOnlineChkDlyTm	:= ADR(tyNtParamCurr.tLFLeaderOnlineChkDlyTm);
	p_NtParamLFLeaderSetTmOffDlyTm	:= ADR(tyNtParamCurr.tLFLeaderSetTmOffDlyTm);

	p_NtParamLFFollowerProgNm		:= ADR(tyNtParamCurr.sLFFollowerProgNm);

	p_NtParamFollower1ProgNm		:= ADR(tyNtParamCurr.sFollower1ProgNm);

	p_NtParamLCSProgNm				:= ADR(tyNtParamCurr.sLCSProgNm);

	p_NtParamLCSMngRcpProgNm		:= ADR(tyNtParamCurr.sLCSMngRcpProgNm);

	p_NtParamLCSLFProgNm			:= ADR(tyNtParamCurr.sLCSLFProgNm);

	p_NtParamProdRcpMinWidth		:= ADR(tyNtParamCurr.tyProdRcpWidthLmt.diMin);
	p_NtParamProdRcpMaxWidth		:= ADR(tyNtParamCurr.tyProdRcpWidthLmt.diMax);
	p_NtParamProdRcpMinMcMod		:= ADR(tyNtParamCurr.tyProdRcpMcModLmt.diMin);
	p_NtParamProdRcpMaxMcMod		:= ADR(tyNtParamCurr.tyProdRcpMcModLmt.diMax);
	p_NtParamProdRcpMinFlippedBrd	:= ADR(tyNtParamCurr.tyProdRcpFlippedBrdLmt.diMin);
	p_NtParamProdRcpMaxFlippedBrd	:= ADR(tyNtParamCurr.tyProdRcpFlippedBrdLmt.diMax);

	// UI Direction L o R / R to L
	p_NtParamUIConvDirRL			:= ADR(tyNtParamCurr.bUIConvDirRL);

	//DBA on Right Sensor
	p_NtParamProjDBAOnRgtSen 		:=ADR(tyNtParamCurr.bProjDBAOnRgtSen);

	//LF new
	p_NtParamLFWidth2Prep			:= ADR(tyNtParamCurr.bLFProdWidth2Prep);
	p_NtParamLFFllowerOnlineChkDlyTm:= ADR(tyNtParamCurr.tLFFollowerOnlineChkDlyTm);

	//machine safety US/DS signal // ADD
	p_NTParamUnlockCovPrep			:= ADR(tyNtParamCurr.bUnlockCoverPrep);
	p_NTParamMachineSafetySig		:= ADR(tyNtParamCurr.bUSDSMachineSafetySig);

	//InvertOnce & InvertTwice_2023_0032B01
	p_NtParamProjInvertOncePrep		:= ADR(tyNtParamCurr.bProjInvertOncePrep);
	p_NtParamProjInvertTwicePrep	:= ADR(tyNtParamCurr.bProjInvertTwicePrep);
	p_NtParamUSExtSMEMA2Prep		:= ADR(tyNtParamCurr.bUSExtSMEMA2Prep);
	p_NtParamUSSMEMA2ProgNm			:= ADR(tyNtParamCurr.sUSSMEMA2ProgNm);
	p_NtParamUSSMEMA2RstDlyTm		:= ADR(tyNtParamCurr.tUSSMEMA2RstDlyTm);
	p_NtParamUSSMEMA2SigInChkTm		:= ADR(tyNtParamCurr.tUSSMEMA2SigInChkTm);
	p_NtParamProjRtrnBrdConvDir		:= ADR(tyNtParamCurr.eProjRtrnBrdConvDir);

	p_NtParamProjChinesePrep		:= ADR(tyNtParamCurr.bChinesePrep);
	p_NtParamProjGermanPrep			:= ADR(tyNtParamCurr.bGemanPrep);

	//Rmt Hermes
	p_NtParamHermesInput            := ADR(tyNtParamCurr.iInput);//Total Input = How many inlet
	p_NtParamHermesOutput           := ADR(tyNtParamCurr.iOutput);//Total Outlet  = How many outlet

	//Svy Hermes
	p_NtParamHermesSvyPrep			:= ADR(tyNtParamCurr.bHermesSvyPrep);
	p_NtParamDSHermesRetainFileNm	:= ADR(tyNtParamCurr.sDSHermesRetainFileNm);
	(* Always Change If Project Change *)

END_PROGRAM
```

### UsrMgmt.typ - Do Not Change!!!
```iecst
(*2019-05-04*)
(**)
(*Action*)

TYPE
	eUsrMgmtAction :
		(
		UsrMgmtActIdle,
		UsrMgmtActCreateDir,
		UsrMgmtActLogin,
		UsrMgmtActBypassLogin,
		UsrMgmtActLogout,
		UsrMgmtActAdd,
		UsrMgmtActEdit,
		UsrMgmtActDel,
		UsrMgmtActSaveAccessRight,
		UsrMgmtActReadData
		);
END_TYPE

(**)
(*Data*)

TYPE
	tyUsrMgmtParam : 	STRUCT
		sUsrNm : STRING[30];
		sPw : STRING[30];
		eUsrLvl : eUsrMgmtAutLvl;
	END_STRUCT;
	eUsrMgmtAutLvl :
		(
		UsrMgmtLvl1,
		UsrMgmtLvl2,
		UsrMgmtLvl3,
		UsrMgmtAdmin,
		UsrMgmtNtEngr,
		UsrMgmtNtAdmin
		);
	tyUsrMgmtAccessRight : 	STRUCT
		bOpt : BOOL;
		bProdSel : BOOL;
		bMagSel : BOOL;
		bMcInfo : BOOL;
		bAlm : BOOL;
		bBffrInfo : BOOL;
		bOvenInfo : BOOL;
		bMagInfo : BOOL;
		bLFCtrl : BOOL;
		bManual : BOOL;
		bManualFBOnly : BOOL;
		bSimulation : BOOL;
		bProdSet : BOOL;
		bMagSet : BOOL;
		bMcSet : BOOL;
		bLang : BOOL;
		bUsrMgmt : BOOL;
		bLFSet : BOOL;
		bChgParam : BOOL;
		sNm : STRING[30];
	END_STRUCT;
	tyUsrMgmtFullDat : 	STRUCT
		a_tyAllList : ARRAY[1..c_udiUsrMgmtMax]OF tyUsrMgmtParam;
		tyAccessRightLvl1 : tyUsrMgmtAccessRight := (bOpt:=TRUE,bProdSel:=TRUE,bMcInfo:=TRUE,bAlm:=TRUE,bLFCtrl:=TRUE);
		tyAccessRightLvl2 : tyUsrMgmtAccessRight := (bOpt:=TRUE,bProdSel:=TRUE,bMagSel:=TRUE,bMcInfo:=TRUE,bAlm:=TRUE,bBffrInfo:=TRUE,bOvenInfo:=TRUE,bMagInfo:=TRUE,bLFCtrl:=TRUE,bProdSet:=TRUE,bChgParam:=TRUE,sNm:='Line Leader');
		tyAccessRightLvl3 : tyUsrMgmtAccessRight := (bOpt:=TRUE,bProdSel:=TRUE,bMagSel:=TRUE,bMcInfo:=TRUE,bAlm:=TRUE,bBffrInfo:=TRUE,bOvenInfo:=TRUE,bMagInfo:=TRUE,bLFCtrl:=TRUE,bManual:=TRUE,bSimulation:=TRUE,bProdSet:=TRUE,bMagSet:=TRUE,bMcSet:=TRUE,bLang:=TRUE,bUsrMgmt:=TRUE,bLFSet:=TRUE,bChgParam:=TRUE,sNm:='Technician');
	END_STRUCT;
END_TYPE
```

### UsrMgmt.var - Change By Project
```iecst
(*2019-05-08*)
(**)
(*Constant*)
VAR CONSTANT
	c_udiUsrMgmtMax : UDINT := 50;
END_VAR
(**)
(*Action & State & Status*)
VAR
	p_UsrMgmtStat : UDINT;
	p_UsrMgmtStatus : UDINT;
	p_UsrMgmtStatTxt : UDINT;
END_VAR
(**)
(*Alarm*)
VAR
	p_UsrMgmtAlmData : UDINT;
END_VAR
(**)
(*Output*)
VAR
	p_UsrMgmtCurrAccessRight : UDINT;
	p_UsrMgmtCurrUsr : UDINT;
	p_UsrMgmtFullData : UDINT;
	p_UsrMgmtAllList : UDINT;
	p_UsrMgmtAccessRightLvl1 : UDINT;
	p_UsrMgmtAccessRightLvl2 : UDINT;
	p_UsrMgmtAccessRightLvl3 : UDINT;
	p_UsrMgmtLvl2List : UDINT;
	p_UsrMgmtLvl3List : UDINT;
	p_UsrMgmtAdminList : UDINT;
	p_UsrMgmtLastAdmin : UDINT;
	p_UsrMgmtUnableDelete : UDINT;
	p_UsrMgmtLoginSuccess : UDINT;
	p_UsrMgmtNmExist : UDINT;
	p_UsrMgmtNmNotExist : UDINT;
	p_UsrMgmtPwMismatch : UDINT;
	p_UsrMgmtNmEmpty : UDINT;
	p_UsrMgmtListFull : UDINT;
	p_UsrMgmtFileNotFound : UDINT;
END_VAR
```

### Program Logical/UsrMgmt/UsrMgmt (IEC) - 1.00.0 - NtRecipe v5.00.0 , NtFileIO v5.00.0 (2018-12-04)

#### InputRef.var
```iecst
(*2019-05-04*)
(**)
(*General*)
VAR
	p_eAct : REFERENCE TO eUsrMgmtAction;
	p_udiMax : REFERENCE TO UDINT;
	p_udiRstErr : REFERENCE TO UDINT;
END_VAR
(**)
(*Configuration*)
VAR
	p_tyInfoIn : REFERENCE TO tyUsrMgmtParam;
	p_tyAccessRightLvl1 : REFERENCE TO tyUsrMgmtAccessRight;
	p_tyAccessRightLvl2 : REFERENCE TO tyUsrMgmtAccessRight;
	p_tyAccessRightLvl3 : REFERENCE TO tyUsrMgmtAccessRight;
	p_sProgNm : REFERENCE TO STRING[15];
	p_bNtSettingsLoadDone : REFERENCE TO BOOL;
END_VAR
```

#### Local.var
```iecst
(*2019-05-04*)
(**)
(*Local Action, State & Status*)
VAR
	eAct : eUsrMgmtAction := UsrMgmtActIdle;
	eStat : eUsrMgmtAction := UsrMgmtActIdle;
	eStatus : eFBStatus := Idle;
	udiStatus : UDINT := 0;
	sStatTxt : STRING[200] := '';
	a_sStatText : ARRAY[0..50] OF STRING[200] := ['Idling','Creating Directory','Logging In','Bypass Logging','Logging Out','Adding New User','Editing User Data','Deleting User','Saving Access Right','Reading Data',41('')];
END_VAR
(**)
(*Local Alarm*)
VAR
	tyAlmData : tyAlmDat;
	a_tyAlmText : ARRAY[10000..10099] OF tyAlmTxt := [(sAlmText:='Create User Folder Error',sRcyText:='Unable To Create User Folder. Please Contact Nutek For A Possible Solution'),(sAlmText:='Create Private Folder Error',sRcyText:='Unable To Create Private Folder. Please Contact Nutek For A Possible Solution'),(sAlmText:='Create UserMgmt Folder Error',sRcyText:='Unable To Create UserMgmt Folder. Please Contact Nutek For A Possible Solution'),(0),(sAlmText:='File Open Error While Adding New User',sRcyText:='An Error Was Encountered While Trying To Open File. Please Contact Nutek For A Possible Solution.'),(sAlmText:='File Create Error While Adding New User',sRcyText:='An Error Was Encountered While Trying To Create File. Please Contact Nutek For A Possible Solution.'),(sAlmText:='File Write Error While Adding New User',sRcyText:='An Error Was Encountered While Trying To Write File. Please Contact Nutek For A Possible Solution.'),(sAlmText:='File Close Error While Adding New User',sRcyText:='An Error Was Encountered While Trying To Close File. Please Contact Nutek For A Possible Solution.'),(sAlmText:='Directory Does Not Exist While Adding New User',sRcyText:='The Directory Does Not Exist.Please Contact Nutek For A Possible Solution.'),(sAlmText:='File Open Error While Saving Access Right',sRcyText:='An Error Was Encountered While Trying To Open File. Please Contact Nutek For A Possible Solution.'),(sAlmText:='File Create Error While Saving Access Right',sRcyText:='An Error Was Encountered While Trying To Create File. Please Contact Nutek For A Possible Solution.'),(sAlmText:='File Write Error While Saving Access Right',sRcyText:='An Error Was Encountered While Trying To Write File. Please Contact Nutek For A Possible Solution.'),(sAlmText:='File Close Error While Saving Access Right',sRcyText:='An Error Was Encountered While Trying To Close File. Please Contact Nutek For A Possible Solution.'),(sAlmText:='Directory Does Not Exist While Saving Access Right',sRcyText:='The Directory Does Not Exist.Please Contact Nutek For A Possible Solution.'),(sAlmText:='File Open Error While Editing User',sRcyText:='An Error Was Encountered While Trying To Open File. Please Contact Nutek For A Possible Solution.'),(sAlmText:='File Create Error While Editing User',sRcyText:='An Error Was Encountered While Trying To Create File. Please Contact Nutek For A Possible Solution.'),(sAlmText:='File Write Error While Editing User',sRcyText:='An Error Was Encountered While Trying To Write File. Please Contact Nutek For A Possible Solution.'),(sAlmText:='File Close Error While Editing User',sRcyText:='An Error Was Encountered While Trying To Close File. Please Contact Nutek For A Possible Solution.'),(sAlmText:='Directory Does Not Exist While Editing User',sRcyText:='The Directory Does Not Exist.Please Contact Nutek For A Possible Solution.'),5((0)),(sAlmText:='File Open Error While Deleting User',sRcyText:='An Error Was Encountered While Trying To Open File. Please Contact Nutek For A Possible Solution.'),(sAlmText:='File Create Error While Deleting User',sRcyText:='An Error Was Encountered While Trying To Create File. Please Contact Nutek For A Possible Solution.'),(sAlmText:='File Write Error While Deleting User',sRcyText:='An Error Was Encountered While Trying To Write File. Please Contact Nutek For A Possible Solution.'),(sAlmText:='File Close Error While Deleting User',sRcyText:='An Error Was Encountered While Trying To Close File. Please Contact Nutek For A Possible Solution.'),(sAlmText:='Directory Does Not Exist While Deleting User',sRcyText:='The Directory Does Not Exist.Please Contact Nutek For A Possible Solution.'),5((0)),(sAlmText:='File Open Error While Getting User List',sRcyText:='An Error Was Encountered While Trying To Open File. Please Contact Nutek For A Possible Solution.'),(sAlmText:='File Read Error While Getting User List',sRcyText:='An Error Was Encountered While Trying To Read File. Please Contact Nutek For A Possible Solution.'),(sAlmText:='File Close Error While Getting User List',sRcyText:='An Error Was Encountered While Trying To Close File. Please Contact Nutek For A Possible Solution.'),3(0),60((0))];
END_VAR
(**)
(*Local Output*)
VAR
	tyCurrAccessRight : tyUsrMgmtAccessRight;
	tyCurrUsr : tyUsrMgmtParam;
	tyFullData : tyUsrMgmtFullDat;
	a_tyLvl2List : ARRAY[1..c_udiUsrMgmtMax] OF tyUsrMgmtParam;
	a_tyLvl3List : ARRAY[1..c_udiUsrMgmtMax] OF tyUsrMgmtParam;
	a_tyAdminList : ARRAY[1..c_udiUsrMgmtMax] OF tyUsrMgmtParam;
	bLastAdmin : BOOL := TRUE;
	bUnableDelete : BOOL;
	bLoginSuccess : BOOL;
	bNmExist : BOOL;
	bNmNotExist : BOOL;
	bPwMismatch : BOOL;
	bNmEmpty : BOOL;
	bListFull : BOOL;
	bFileNotFound : BOOL;
END_VAR
(**)
(*Local Input*)
VAR
	udiRstErr : UDINT := 0;
	tyInfoIn : tyUsrMgmtParam;
	tyAccessRightLvl1 : tyUsrMgmtAccessRight;
	tyAccessRightLvl2 : tyUsrMgmtAccessRight;
	tyAccessRightLvl3 : tyUsrMgmtAccessRight;
	sProgNm : STRING[15] := 'UsrMgmt';
	bNtSettingsLoadDone : BOOL := TRUE;
END_VAR
(**)
(*Local*)
VAR
	bRstErr : BOOL;
	udiRstErrOld : UDINT;
	bInitDone : BOOL;
	bInitialDone : BOOL;
	usiStep : USINT := 0;
	udiAddStatus : UDINT;
	tyAccessRightAdmin : tyUsrMgmtAccessRight := (bOpt:=TRUE,bProdSel:=TRUE,bMagSel:=TRUE,bMcInfo:=TRUE,bAlm:=TRUE,bBffrInfo:=TRUE,bOvenInfo:=TRUE,bMagInfo:=TRUE,bLFCtrl:=TRUE,bManual:=TRUE,bSimulation:=TRUE,bProdSet:=TRUE,bMagSet:=TRUE,bMcSet:=TRUE,bLang:=TRUE,bUsrMgmt:=TRUE,bLFSet:=TRUE,bChgParam:=TRUE,sNm:='Admin');
	fbDirCreate1 : fbDirCreate;
	fbDirCreate2 : fbDirCreate;
	fbDirCreate3 : fbDirCreate;
	fbFileRead1 : fbFileFullReadEncry;
	fbFileWrite1 : fbFileFullWriteEncry;
	tyFullDataTemp : tyUsrMgmtFullDat;
	tyInfoOut : tyUsrMgmtParam;
	udi : UDINT;
	udiCnt : UDINT;
	udiCnt1 : UDINT;
	udiCnt2 : UDINT;
	udiModuleNum : UINT := 5351;
END_VAR
```

#### Act_Action.st
```iecst
(** 2019-03-25 **)
ACTION Act_Action:

	//Reset Error
	IF (eStatus = Error) AND bRstErr THEN
		p_eAct	:= UsrMgmtActIdle;
		eStat	:= UsrMgmtActIdle;
	END_IF

	//Reset Done
	IF eStatus = Done AND p_eAct = UsrMgmtActIdle THEN
		eStat	:= UsrMgmtActIdle;
	END_IF

	//Set p_eAct
	IF eStatus = Idle THEN
		eStat	:= p_eAct;
	END_IF

END_ACTION
```

#### Act_Alarm.st
```iecst
(** 2019-03-25 **)
ACTION Act_Alarm:

	//Error
	IF EDGEPOS(eStatus = Error) THEN

		tyAlmData.sProgNm		:= p_sProgNm;
		tyAlmData.udiCode		:= udiStatus;
		tyAlmData.eSeverity		:= AlmSeverityError;
		tyAlmData.udiRunTime	:= tyAlmData.udiRunTime + 1;
		tyAlmData.bAlm			:= TRUE;
		tyAlmData.udiModuleNum  := udiModuleNum;
		g_sUsrMgmtProgNm		:= p_sProgNm;

		//Get Error Message
		IF tyAlmData.udiCode < 10000 OR tyAlmData.udiCode > 10099 THEN
			tyAlmData.sAlmMsg	:= 'Unknown';
			tyAlmData.sRcyMsg	:= 'Unknown';
		ELSE
			tyAlmData.sAlmMsg	:= a_tyAlmText[tyAlmData.udiCode].sAlmText;
			tyAlmData.sRcyMsg	:= a_tyAlmText[tyAlmData.udiCode].sRcyText;
		END_IF

		sStatTxt	:= tyAlmData.sAlmMsg;

	ELSIF bRstErr AND (tyAlmData.udiCode <> 0) THEN

		tyAlmData.udiCode	:= 0;
		tyAlmData.eSeverity	:= AlmSeverityNA;
		tyAlmData.sAlmMsg	:= '';
		tyAlmData.sRcyMsg	:= '';
		tyAlmData.bAlm			:= FALSE;
		sStatTxt	:= a_sStatText[eStat];

	END_IF

END_ACTION
```

#### Act_InitGlobal.st
```iecst
(** 2019-03-25 **)
ACTION Act_InitGlobal:

	(* Always Change If Project Change *)

	//Pass Data To Link
	p_bLinkStartupRun ACCESS p_StartupRun;

	//Pass Data To Internal Use
	p_udiRstErr ACCESS p_RstErrReset;
	p_tyInfoIn ACCESS p_UIUsrMgmtInfoIn;
	p_tyAccessRightLvl1 ACCESS p_UIUsrMgmtAccessRightLvl1Wr;
	p_tyAccessRightLvl2 ACCESS p_UIUsrMgmtAccessRightLvl2Wr;
	p_tyAccessRightLvl3 ACCESS p_UIUsrMgmtAccessRightLvl3Wr;
	p_sProgNm ACCESS p_NtParamUsrMgmtProgNm;
	p_bNtSettingsLoadDone ACCESS p_StartupNtSettingsLoadDone;

	(* Always Change If Project Change *)

END_ACTION
```

#### Act_Initial.st
```iecst
(** 2019-05-04 **)
ACTION Act_Initial:

	//Initial
	sStatTxt	:= a_sStatText[eStat];

	fbDirCreate1.sDevice	:= 'F';
	fbDirCreate1.sDirName	:= 'User';
	fbDirCreate1(bEn := FALSE);

	fbDirCreate2.sDevice	:= 'F';
	fbDirCreate2.sDirName	:= 'Private';
	fbDirCreate2(bEn := FALSE);

	fbDirCreate3.sDevice	:= 'User';
	fbDirCreate3.sDirName	:= 'UserMgmt';
	fbDirCreate3(bEn := FALSE);

	fbFileRead1.sDevice			:= 'CustomerUser';
	fbFileRead1.sFile			:= 'User.dat';
	fbFileRead1.udiOffset		:= 0;
	fbFileRead1.p_Dest			:= ADR(tyFullData);
	fbFileRead1.udiLen			:= SIZEOF(tyFullData);
	fbFileRead1.usiEncryptCode	:= 130;
	fbFileRead1(bEn := FALSE);

	fbFileWrite1.sDevice		:= 'CustomerUser';
	fbFileWrite1.sFile			:= 'User.dat';
	fbFileWrite1.udiOffset		:= 0;
	fbFileWrite1.p_Src			:= ADR(tyFullDataTemp);
	fbFileWrite1.udiLen			:= SIZEOF(tyFullDataTemp);
	fbFileWrite1.udiOption		:= 0;
	fbFileWrite1.usiEncryptCode	:= 130;
	fbFileWrite1(bEn := FALSE);

END_ACTION
```

#### Act_InitLocal.st
```iecst
(** 2019-05-04 **)
ACTION Act_InitLocal:

	//Input Reference Link To Local Variable
	p_eAct ACCESS ADR(eAct);
	p_udiMax ACCESS ADR(c_udiUsrMgmtMax);
	p_udiRstErr ACCESS ADR(udiRstErr);
	p_tyInfoIn ACCESS ADR(tyInfoIn);
	p_tyAccessRightLvl1 ACCESS ADR(tyAccessRightLvl1);
	p_tyAccessRightLvl2 ACCESS ADR(tyAccessRightLvl2);
	p_tyAccessRightLvl3 ACCESS ADR(tyAccessRightLvl3);
	p_sProgNm ACCESS ADR(sProgNm);
	p_bNtSettingsLoadDone ACCESS ADR(bNtSettingsLoadDone);

END_ACTION
```

#### Act_LinkAction.st
```iecst
(** 2019-03-29 **)
ACTION Act_LinkAction:

	IF p_bLinkStartupRun = TRUE THEN
		p_eAct ACCESS p_StartupUsrMgmtAct;
	ELSE
		p_eAct ACCESS p_UIUsrMgmtAct;
	END_IF

END_ACTION
```

#### Act_Main.st
```iecst
(** 2019-05-04 **)
ACTION Act_Main:

	//Main
	CASE eStat OF

		UsrMgmtActIdle:
			IF eStatus <> Idle THEN	//Reset Data
				//Private
				fbDirCreate1(bEn := FALSE);
				fbDirCreate2(bEn := FALSE);
				fbDirCreate3(bEn := FALSE);
				fbFileRead1(bEn := FALSE);
				fbFileWrite1(bEn := FALSE);
				usiStep			:= 0;
				udiAddStatus	:= 0;

				bListFull			:= FALSE;
				bLoginSuccess		:= FALSE;
				bNmEmpty			:= FALSE;
				bNmExist			:= FALSE;
				bNmNotExist			:= FALSE;
				bPwMismatch			:= FALSE;
				bFileNotFound		:= FALSE;
				bUnableDelete		:= FALSE;

				sStatTxt	:= a_sStatText[eStat];

			END_IF

			eStatus	:= Idle;

		UsrMgmtActCreateDir:
			IF eStatus = Idle OR eStatus = Busy THEN

				eStatus	:= Busy;

				sStatTxt	:= a_sStatText[eStat];

				CASE usiStep OF
					0:
						fbDirCreate1(bEn := TRUE);
						IF fbDirCreate1.udiStatus = 0 THEN
							usiStep	:= 1;
						ELSIF fbDirCreate1.udiStatus < 65534 THEN
							eStatus	:= Error;

							IF fbDirCreate1.udiStatus = 1908 THEN
								udiStatus	:= 10000;	//Create User Folder Error
							ELSE
								udiStatus	:= fbDirCreate1.udiStatus;
							END_IF
						END_IF

					1:
						fbDirCreate2(bEn := TRUE);
						IF fbDirCreate2.udiStatus = 0 THEN
							usiStep	:= 2;
						ELSIF fbDirCreate2.udiStatus < 65534 THEN
							eStatus	:= Error;

							IF fbDirCreate2.udiStatus = 1908 THEN
								udiStatus	:= 10001;	//Create Private Folder Error
							ELSE
								udiStatus	:= fbDirCreate2.udiStatus;
							END_IF
						END_IF

					2:
						fbDirCreate3(bEn := TRUE);
						IF fbDirCreate3.udiStatus = 0 THEN
							eStatus	:= Done;
						ELSIF fbDirCreate3.udiStatus < 65534 THEN
							eStatus	:= Error;

							IF fbDirCreate3.udiStatus = 1908 THEN
								udiStatus	:= 10002;	//Create UserMgmt Folder Error
							ELSE
								udiStatus	:= fbDirCreate3.udiStatus;
							END_IF
						END_IF

				END_CASE

			END_IF

		UsrMgmtActLogin:
			IF eStatus = Idle OR eStatus = Busy THEN

				sStatTxt	:= a_sStatText[eStat];

				bNmNotExist	:= (fRecipeGetInfo(p_tyInfoIn.sUsrNm , ADR(tyInfoOut) , ADR(tyFullData.a_tyAllList) , SIZEOF(tyFullData.a_tyAllList[1]) , ADR(tyFullData.a_tyAllList[1].sUsrNm) , SIZEOF(tyFullData.a_tyAllList[1].sUsrNm) , p_udiMax)) = 0;

				IF (bNmNotExist = FALSE) THEN

					IF (p_tyInfoIn.sPw = tyInfoOut.sPw) THEN
						bLoginSuccess	:= TRUE;
						bPwMismatch		:= FALSE;
						tyCurrUsr		:= tyInfoOut;

						IF tyCurrUsr.eUsrLvl = UsrMgmtLvl2 THEN

							tyCurrAccessRight			:= tyFullData.tyAccessRightLvl2;
							tyCurrAccessRight.bUsrMgmt	:= FALSE;

							IF tyCurrAccessRight.sNm = '' THEN
								tyCurrAccessRight.sNm	:= 'Level2';
							END_IF

						ELSIF tyCurrUsr.eUsrLvl = UsrMgmtLvl3 THEN

							tyCurrAccessRight			:= tyFullData.tyAccessRightLvl3;
							tyCurrAccessRight.bUsrMgmt	:= FALSE;

							IF tyCurrAccessRight.sNm = '' THEN
								tyCurrAccessRight.sNm	:= 'Level3';
							END_IF

						ELSIF tyCurrUsr.eUsrLvl = UsrMgmtAdmin THEN

							tyCurrAccessRight			:= tyAccessRightAdmin;

						END_IF

					ELSE
						bLoginSuccess				:= FALSE;
						bPwMismatch					:= TRUE;
						tyCurrUsr.sUsrNm			:= '';
						tyCurrUsr.sPw				:= '';
						tyCurrUsr.eUsrLvl			:= UsrMgmtLvl1;
						tyCurrAccessRight			:= tyFullData.tyAccessRightLvl1;
						tyCurrAccessRight.bUsrMgmt	:= FALSE;

						IF tyCurrAccessRight.sNm = '' THEN
							tyCurrAccessRight.sNm	:= 'Level1';
						END_IF

					END_IF

				ELSE
					bLoginSuccess				:= FALSE;
					bPwMismatch					:= FALSE;
					tyCurrUsr.sUsrNm			:= '';
					tyCurrUsr.sPw				:= '';
					tyCurrUsr.eUsrLvl			:= UsrMgmtLvl1;
					tyCurrAccessRight			:= tyFullData.tyAccessRightLvl1;
					tyCurrAccessRight.bUsrMgmt	:= FALSE;

					IF tyCurrAccessRight.sNm = '' THEN
						tyCurrAccessRight.sNm	:= 'Level1';
					END_IF

				END_IF

				eStatus	:= Done;

			END_IF

		UsrMgmtActBypassLogin:
			IF eStatus = Idle OR eStatus = Busy THEN

				sStatTxt	:= a_sStatText[eStat];

				bLoginSuccess		:= TRUE;
				tyCurrUsr.sUsrNm	:= 'User Bypass';
				tyCurrUsr.sPw		:= '';
				tyCurrUsr.eUsrLvl	:= UsrMgmtAdmin;
				tyCurrAccessRight	:= tyAccessRightAdmin;

				eStatus	:= Done;

			END_IF

		UsrMgmtActLogout:
			IF eStatus = Idle OR eStatus = Busy THEN

				sStatTxt	:= a_sStatText[eStat];

				tyCurrUsr.sUsrNm			:= '';
				tyCurrUsr.sPw				:= '';
				tyCurrUsr.eUsrLvl			:= UsrMgmtLvl1;
				tyCurrAccessRight			:= tyFullData.tyAccessRightLvl1;
				tyCurrAccessRight.bUsrMgmt	:= FALSE;

				IF tyCurrAccessRight.sNm = '' THEN
					tyCurrAccessRight.sNm	:= 'Level1';
				END_IF

				eStatus	:= Done;

			END_IF

		UsrMgmtActAdd:
			IF eStatus = Idle OR eStatus = Busy THEN

				eStatus	:= Busy;

				sStatTxt	:= a_sStatText[eStat];

				CASE usiStep OF
					0:	//Add User
						udiAddStatus	:= fRecipeAdd(ADR(p_tyInfoIn) , ADR(tyFullDataTemp.a_tyAllList) , SIZEOF(tyFullDataTemp.a_tyAllList[1]) , ADR(tyFullDataTemp.a_tyAllList[1].sUsrNm) , SIZEOF(tyFullDataTemp.a_tyAllList[1].sUsrNm) , p_udiMax);

						IF udiAddStatus = 1600 THEN	//Recipe Name Empty
							bNmEmpty	:= TRUE;
							eStatus		:= Done;

						ELSIF udiAddStatus = 1601 THEN	//Recipe Full
							bListFull	:= TRUE;
							eStatus		:= Done;

						ELSIF udiAddStatus = 1602 THEN	//Recipe Name Exist
							bNmExist	:= TRUE;
							eStatus		:= Done;

						ELSIF udiAddStatus = 0 THEN	//OK
							usiStep	:= 1;

						END_IF

					1:	//Write Into File
						fbFileWrite1(bEn := TRUE);

						IF fbFileWrite1.udiStatus = 0 THEN
							tyFullData.a_tyAllList	:= tyFullDataTemp.a_tyAllList;

							IF p_tyInfoIn.eUsrLvl = UsrMgmtLvl2 THEN
								udiCnt	:= 1;
								memset(ADR(a_tyLvl2List) , 0 , SIZEOF(a_tyLvl2List));

								FOR udi := 1 TO p_udiMax DO
									IF tyFullData.a_tyAllList[udi].eUsrLvl = UsrMgmtLvl2 THEN
										a_tyLvl2List[udiCnt]	:= tyFullData.a_tyAllList[udi];
										udiCnt					:= udiCnt + 1;
									END_IF
								END_FOR

							ELSIF p_tyInfoIn.eUsrLvl = UsrMgmtLvl3 THEN
								udiCnt	:= 1;
								memset(ADR(a_tyLvl3List) , 0 , SIZEOF(a_tyLvl3List));

								FOR udi := 1 TO p_udiMax DO
									IF tyFullData.a_tyAllList[udi].eUsrLvl = UsrMgmtLvl3 THEN
										a_tyLvl3List[udiCnt]	:= tyFullData.a_tyAllList[udi];
										udiCnt					:= udiCnt + 1;
									END_IF
								END_FOR

							ELSIF p_tyInfoIn.eUsrLvl = UsrMgmtAdmin THEN
								udiCnt		:= 1;
								bLastAdmin	:= TRUE;
								memset(ADR(a_tyAdminList) , 0 , SIZEOF(a_tyAdminList));

								FOR udi := 1 TO p_udiMax DO
									IF tyFullData.a_tyAllList[udi].eUsrLvl = UsrMgmtAdmin THEN
										a_tyAdminList[udiCnt]	:= tyFullData.a_tyAllList[udi];
										bLastAdmin				:= udiCnt = 1;
										udiCnt					:= udiCnt + 1;
									END_IF
								END_FOR

							END_IF

							eStatus	:= Done;

						ELSIF fbFileWrite1.udiStatus < 65534 THEN
							tyFullDataTemp.a_tyAllList	:= tyFullData.a_tyAllList;
							eStatus						:= Error;

							IF fbFileWrite1.udiStatus = 1900 THEN
								udiStatus	:= 10004;	//File Open Error While Adding New User
							ELSIF fbFileWrite1.udiStatus = 1901 THEN
								udiStatus	:= 10005;	//File Create Error While Adding New User
							ELSIF fbFileWrite1.udiStatus = 1903 THEN
								udiStatus	:= 10006;	//File Write Error While Adding New User
							ELSIF fbFileWrite1.udiStatus = 1904 THEN
								udiStatus	:= 10007;	//File Close Error While Adding New User
							ELSIF fbFileWrite1.udiStatus = 1914 THEN
								udiStatus	:= 10008;	//Directory Does Not Exist While Adding New User
							ELSE
								udiStatus	:= fbFileWrite1.udiStatus;
							END_IF
						END_IF

				END_CASE

			END_IF

		UsrMgmtActEdit:
			IF eStatus = Idle OR eStatus = Busy THEN

				eStatus	:= Busy;

				sStatTxt	:= a_sStatText[eStat];

				CASE usiStep OF
					0:	//Edit User
						udiAddStatus	:= fRecipeAddEdit(ADR(p_tyInfoIn) , ADR(tyFullDataTemp.a_tyAllList) , SIZEOF(tyFullDataTemp.a_tyAllList[1]) , ADR(tyFullDataTemp.a_tyAllList[1].sUsrNm) , SIZEOF(tyFullDataTemp.a_tyAllList[1].sUsrNm) , p_udiMax);

						IF udiAddStatus = 1600 THEN	//Recipe Name Empty
							bNmEmpty	:= TRUE;
							eStatus		:= Done;

						ELSIF udiAddStatus = 1601 THEN	//Recipe Full
							bListFull	:= TRUE;
							eStatus		:= Done;

						ELSIF udiAddStatus = 0 THEN	//OK
							usiStep	:= 1;

						END_IF

					1:	//Write Into File
						fbFileWrite1(bEn := TRUE);

						IF fbFileWrite1.udiStatus = 0 THEN
							tyFullData.a_tyAllList	:= tyFullDataTemp.a_tyAllList;

							udiCnt			:= 1;
							udiCnt1			:= 1;
							udiCnt2			:= 1;
							bLastAdmin	:= TRUE;
							memset(ADR(a_tyLvl2List) , 0 , SIZEOF(a_tyLvl2List));
							memset(ADR(a_tyLvl3List) , 0 , SIZEOF(a_tyLvl3List));
							memset(ADR(a_tyAdminList) , 0 , SIZEOF(a_tyAdminList));

							FOR udi := 1 TO p_udiMax DO
								IF tyFullData.a_tyAllList[udi].eUsrLvl = UsrMgmtLvl2 THEN
									a_tyLvl2List[udiCnt]	:= tyFullData.a_tyAllList[udi];
									udiCnt					:= udiCnt + 1;
								ELSIF tyFullData.a_tyAllList[udi].eUsrLvl = UsrMgmtLvl3 THEN
									a_tyLvl3List[udiCnt1]	:= tyFullData.a_tyAllList[udi];
									udiCnt1					:= udiCnt1 + 1;
								ELSIF tyFullData.a_tyAllList[udi].eUsrLvl = UsrMgmtAdmin THEN
									a_tyAdminList[udiCnt2]	:= tyFullData.a_tyAllList[udi];
									bLastAdmin				:= udiCnt2 = 1;
									udiCnt2					:= udiCnt2 + 1;
								END_IF
							END_FOR

							eStatus	:= Done;

						ELSIF fbFileWrite1.udiStatus < 65534 THEN
							tyFullDataTemp.a_tyAllList	:= tyFullData.a_tyAllList;
							eStatus						:= Error;

							IF fbFileWrite1.udiStatus = 1900 THEN
								udiStatus	:= 10014;	//File Open Error While Editing User
							ELSIF fbFileWrite1.udiStatus = 1901 THEN
								udiStatus	:= 10015;	//File Create Error While Editing User
							ELSIF fbFileWrite1.udiStatus = 1903 THEN
								udiStatus	:= 10016;	//File Write Error While Editing User
							ELSIF fbFileWrite1.udiStatus = 1904 THEN
								udiStatus	:= 10017;	//File Close Error While Editing User
							ELSIF fbFileWrite1.udiStatus = 1914 THEN
								udiStatus	:= 10018;	//Directory Does Not Exist While Editing User
							ELSE
								udiStatus	:= fbFileWrite1.udiStatus;
							END_IF
						END_IF

				END_CASE

			END_IF

		UsrMgmtActDel:
			IF eStatus = Idle OR eStatus = Busy THEN

				eStatus	:= Busy;

				sStatTxt	:= a_sStatText[eStat];

				CASE usiStep OF
					0: //Check Whether Admin To Delete
						IF p_tyInfoIn.eUsrLvl = UsrMgmtAdmin THEN
							usiStep	:= 1;
						ELSE
							usiStep	:= 2;
						END_IF

					1:	//Check Last Admin
						IF bLastAdmin = FALSE THEN
							usiStep	:= 2;
						ELSE
							bUnableDelete	:= TRUE;
							eStatus			:= Done;
						END_IF

					2:	//Delete User
						udiAddStatus	:= fRecipeDelete(ADR(p_tyInfoIn) , ADR(tyFullDataTemp.a_tyAllList) , SIZEOF(tyFullDataTemp.a_tyAllList[1]) , ADR(tyFullDataTemp.a_tyAllList[1].sUsrNm) , SIZEOF(tyFullDataTemp.a_tyAllList[1].sUsrNm) , p_udiMax);

						IF udiAddStatus = 1600 THEN	//Recipe Name Empty
							bUnableDelete	:= TRUE;
							bNmEmpty		:= TRUE;
							eStatus			:= Done;

						ELSIF udiAddStatus = 1603 THEN	//Recipe Not Exist
							bUnableDelete	:= TRUE;
							bNmNotExist		:= TRUE;
							eStatus			:= Done;

						ELSIF udiAddStatus = 0 THEN	//OK
							usiStep	:= 3;

						END_IF

					3:	//Write Into File
						fbFileWrite1(bEn := TRUE);

						IF fbFileWrite1.udiStatus = 0 THEN
							tyFullData.a_tyAllList	:= tyFullDataTemp.a_tyAllList;

							IF p_tyInfoIn.eUsrLvl = UsrMgmtLvl2 THEN
								udiCnt	:= 1;
								memset(ADR(a_tyLvl2List) , 0 , SIZEOF(a_tyLvl2List));

								FOR udi := 1 TO p_udiMax DO
									IF tyFullData.a_tyAllList[udi].eUsrLvl = UsrMgmtLvl2 THEN
										a_tyLvl2List[udiCnt]	:= tyFullData.a_tyAllList[udi];
										udiCnt					:= udiCnt + 1;
									END_IF
								END_FOR

							ELSIF p_tyInfoIn.eUsrLvl = UsrMgmtLvl3 THEN
								udiCnt	:= 1;
								memset(ADR(a_tyLvl3List) , 0 , SIZEOF(a_tyLvl3List));

								FOR udi := 1 TO p_udiMax DO
									IF tyFullData.a_tyAllList[udi].eUsrLvl = UsrMgmtLvl3 THEN
										a_tyLvl3List[udiCnt]	:= tyFullData.a_tyAllList[udi];
										udiCnt					:= udiCnt + 1;
									END_IF
								END_FOR

							ELSIF p_tyInfoIn.eUsrLvl = UsrMgmtAdmin THEN
								udiCnt			:= 1;
								bLastAdmin	:= TRUE;
								memset(ADR(a_tyAdminList) , 0 , SIZEOF(a_tyAdminList));

								FOR udi := 1 TO p_udiMax DO
									IF tyFullData.a_tyAllList[udi].eUsrLvl = UsrMgmtAdmin THEN
										a_tyAdminList[udiCnt]	:= tyFullData.a_tyAllList[udi];
										bLastAdmin				:= udiCnt = 1;
										udiCnt					:= udiCnt + 1;
									END_IF
								END_FOR

							END_IF

							eStatus	:= Done;

						ELSIF fbFileWrite1.udiStatus < 65534 THEN
							tyFullDataTemp.a_tyAllList	:= tyFullData.a_tyAllList;
							eStatus						:= Error;

							IF fbFileWrite1.udiStatus = 1900 THEN
								udiStatus	:= 10024;	//File Open Error While Deleting User
							ELSIF fbFileWrite1.udiStatus = 1901 THEN
								udiStatus	:= 10025;	//File Create Error While Deleting User
							ELSIF fbFileWrite1.udiStatus = 1903 THEN
								udiStatus	:= 10026;	//File Write Error While Deleting User
							ELSIF fbFileWrite1.udiStatus = 1904 THEN
								udiStatus	:= 10027;	//File Close Error While Deleting User
							ELSIF fbFileWrite1.udiStatus = 1914 THEN
								udiStatus	:= 10028;	//Directory Does Not Exist While Deleting User
							ELSE
								udiStatus	:= fbFileWrite1.udiStatus;
							END_IF
						END_IF

				END_CASE

			END_IF

		UsrMgmtActSaveAccessRight:
			IF eStatus = Idle OR eStatus = Busy THEN

				eStatus	:= Busy;

				sStatTxt	:= a_sStatText[eStat];

				CASE usiStep OF
					0:	//Save Access Right
						tyFullDataTemp.tyAccessRightLvl1	:= p_tyAccessRightLvl1;
						tyFullDataTemp.tyAccessRightLvl2	:= p_tyAccessRightLvl2;
						tyFullDataTemp.tyAccessRightLvl3	:= p_tyAccessRightLvl3;

						usiStep	:= 1;

					1:	//Write Into File
						fbFileWrite1(bEn := TRUE);

						IF fbFileWrite1.udiStatus = 0 THEN
							tyFullData.tyAccessRightLvl1	:= tyFullDataTemp.tyAccessRightLvl1;
							tyFullData.tyAccessRightLvl2	:= tyFullDataTemp.tyAccessRightLvl2;
							tyFullData.tyAccessRightLvl3	:= tyFullDataTemp.tyAccessRightLvl3;
							eStatus							:= Done;

						ELSIF fbFileWrite1.udiStatus < 65534 THEN
							tyFullDataTemp.tyAccessRightLvl1	:= tyFullData.tyAccessRightLvl1;
							tyFullDataTemp.tyAccessRightLvl2	:= tyFullData.tyAccessRightLvl2;
							tyFullDataTemp.tyAccessRightLvl3	:= tyFullData.tyAccessRightLvl3;
							eStatus								:= Error;

							IF fbFileWrite1.udiStatus = 1900 THEN
								udiStatus	:= 10009;	//File Open Error While Saving Access Right
							ELSIF fbFileWrite1.udiStatus = 1901 THEN
								udiStatus	:= 10010;	//File Create Error While Saving Access Right
							ELSIF fbFileWrite1.udiStatus = 1903 THEN
								udiStatus	:= 10011;	//File Write Error While Saving Access Right
							ELSIF fbFileWrite1.udiStatus = 1904 THEN
								udiStatus	:= 10012;	//File Close Error While Saving Access Right
							ELSIF fbFileWrite1.udiStatus = 1914 THEN
								udiStatus	:= 10013;	//Directory Does Not Exist While Saving Access Right
							ELSE
								udiStatus	:= fbFileWrite1.udiStatus;
							END_IF
						END_IF

				END_CASE

			END_IF

		UsrMgmtActReadData:
			IF eStatus = Idle OR eStatus = Busy THEN

				eStatus	:= Busy;

				sStatTxt	:= a_sStatText[eStat];

				fbFileRead1(bEn := TRUE);
				IF fbFileRead1.udiStatus = 0 THEN
					tyFullDataTemp.a_tyAllList	:= tyFullData.a_tyAllList;

					udiCnt			:= 1;
					udiCnt1			:= 1;
					udiCnt2			:= 1;
					bLastAdmin	:= TRUE;
					memset(ADR(a_tyLvl2List) , 0 , SIZEOF(a_tyLvl2List));
					memset(ADR(a_tyLvl3List) , 0 , SIZEOF(a_tyLvl3List));
					memset(ADR(a_tyAdminList) , 0 , SIZEOF(a_tyAdminList));

					FOR udi := 1 TO p_udiMax DO
						IF tyFullData.a_tyAllList[udi].eUsrLvl = UsrMgmtLvl2 THEN
							a_tyLvl2List[udiCnt]	:= tyFullData.a_tyAllList[udi];
							udiCnt					:= udiCnt + 1;
						ELSIF tyFullData.a_tyAllList[udi].eUsrLvl = UsrMgmtLvl3 THEN
							a_tyLvl3List[udiCnt1]	:= tyFullData.a_tyAllList[udi];
							udiCnt1					:= udiCnt1 + 1;
						ELSIF tyFullData.a_tyAllList[udi].eUsrLvl = UsrMgmtAdmin THEN
							a_tyAdminList[udiCnt2]	:= tyFullData.a_tyAllList[udi];
							bLastAdmin				:= udiCnt2 = 1;
							udiCnt2					:= udiCnt2 + 1;
						END_IF
					END_FOR

					eStatus	:= Done;

				ELSIF fbFileRead1.udiStatus < 65534 THEN
					eStatus		:= Error;

					IF fbFileRead1.udiStatus = 1900 THEN
						udiStatus	:= 10034;	//File Open Error While Getting User List
					ELSIF fbFileRead1.udiStatus = 1902 THEN
						udiStatus	:= 10035;	//File Read Error While Getting User List
					ELSIF fbFileRead1.udiStatus = 1904 THEN
						udiStatus	:= 10036;	//File Close Error While Getting User List
					ELSIF fbFileRead1.udiStatus = 1915 THEN
						eStatus			:= Done;
						bFileNotFound	:= TRUE;
					ELSE
						udiStatus	:= fbFileRead1.udiStatus;
					END_IF
				END_IF

			END_IF

	END_CASE

END_ACTION
```

#### Cyclic.st
```iecst
(** 2019-03-29 **)
PROGRAM _CYCLIC

	IF bInitDone = FALSE THEN
		bInitDone	:= TRUE;

		Act_InitLocal;
		Act_InitGlobal;

	ELSIF bInitialDone = FALSE THEN
		IF p_bNtSettingsLoadDone = TRUE THEN
			bInitialDone	:= TRUE;

			Act_Initial;

		END_IF

	ELSE

		Act_RstErr;
		Act_LinkAction;
		Act_Action;
		Act_Link;
		Act_Main;
		Act_Alarm;

	END_IF

END_PROGRAM
```

#### Init.st
```iecst
(** 2019-05-08 **)
PROGRAM _INIT

	(* Always Change If Project Change *)

	//Pass Address To Global Address For External Use
	//Action, State & Status
	p_UsrMgmtStat		:= ADR(eStat);
	p_UsrMgmtStatus		:= ADR(eStatus);
	p_UsrMgmtStatTxt	:= ADR(sStatTxt);

	//Alarm
	p_UsrMgmtAlmData	:= ADR(tyAlmData);

	//Output
	p_UsrMgmtCurrAccessRight	:= ADR(tyCurrAccessRight);
	p_UsrMgmtCurrUsr			:= ADR(tyCurrUsr);
	p_UsrMgmtFullData			:= ADR(tyFullData);
	p_UsrMgmtAllList			:= ADR(tyFullData.a_tyAllList);
	p_UsrMgmtAccessRightLvl1	:= ADR(tyFullData.tyAccessRightLvl1);
	p_UsrMgmtAccessRightLvl2	:= ADR(tyFullData.tyAccessRightLvl2);
	p_UsrMgmtAccessRightLvl3	:= ADR(tyFullData.tyAccessRightLvl3);
	p_UsrMgmtLvl2List			:= ADR(a_tyLvl2List);
	p_UsrMgmtLvl3List			:= ADR(a_tyLvl3List);
	p_UsrMgmtAdminList			:= ADR(a_tyAdminList);
	p_UsrMgmtLastAdmin			:= ADR(bLastAdmin);
	p_UsrMgmtUnableDelete		:= ADR(bUnableDelete);
	p_UsrMgmtLoginSuccess		:= ADR(bLoginSuccess);
	p_UsrMgmtNmExist			:= ADR(bNmExist);
	p_UsrMgmtNmNotExist			:= ADR(bNmNotExist);
	p_UsrMgmtPwMismatch			:= ADR(bPwMismatch);
	p_UsrMgmtNmEmpty			:= ADR(bNmEmpty);
	p_UsrMgmtListFull			:= ADR(bListFull);
	p_UsrMgmtFileNotFound		:= ADR(bFileNotFound);

	(* Always Change If Project Change *)

END_PROGRAM
```

### SMEMA.typ - Do Not Change!!!
```iecst
(*2018-12-13*)
(**)
(*Action*)

TYPE
	eSMEMAAction :
		(
		SMEMAActIdle,
		SMEMAActRun,
		SMEMAActSetSig,
		SMEMAActSetStatSig,
		SMEMAActRstSig,
		SMEMAActRstStatSig,
		SMEMAActSetAllSig,
		SMEMAActRstAllSig
		);
END_TYPE

(**)

TYPE
	tySMEMAParam : 	STRUCT
		eSelection : eSMEMASelection;
		bStatSigSetGd : BOOL;
	END_STRUCT;
	eSMEMASelection :
		(
		SMEMASelStandard,
		SMEMASelIPC9851,
		SMEMASelIPC9851Ext
		);
END_TYPE
```

### USSMEMA.var - Change By Project
```iecst
(*2019-03-25*)
(**)
(*Action & State & Status*)
VAR
	p_USSMEMAStat : UDINT;
	p_USSMEMAStatus : UDINT;
	p_USSMEMAStatTxt : UDINT;
END_VAR
(**)
(*Alarm*)
VAR
	p_USSMEMAAlmData : UDINT;
END_VAR
(**)
(*Output*)
VAR
	p_USSMEMAUSRdy : UDINT;
	p_USSMEMAUSGdBrdRdy : UDINT;
	p_USSMEMADSRdy : UDINT;
	p_USSMEMATransporting : UDINT;
	p_USSMEMAConvStart : UDINT;
	p_USSMEMAConvStop : UDINT;
	p_USSMEMAUSB : UDINT;
	p_USSMEMATimer : UDINT;
	p_USSMEMAVirtual : UDINT;
END_VAR
```

### Program Logical/SMEMA/USSMEMA (IEC, version 1.00.0) - 1.00.0 - NtSMEMA v5.00.0

#### Init.st - Change By Project
```iecst
(** 2019-03-25 **)
PROGRAM _INIT

	(* Always Change If Project Change *)

	//Pass Address To Global Address For External Use
	//Action, State & Status
	p_USSMEMAStat		:= ADR(eStat);
	p_USSMEMAStatus		:= ADR(eStatus);
	p_USSMEMAStatTxt	:= ADR(sStatTxt);

	//Alarm
	p_USSMEMAAlmData	:= ADR(tyAlmData);

	//Output
	p_USSMEMAUSRdy			:= ADR(bUSRdy);
	p_USSMEMAUSGdBrdRdy		:= ADR(bUSGdBrdRdy);
	p_USSMEMADSRdy			:= ADR(bDSRdy);
	p_USSMEMATransporting	:= ADR(bTransporting);
	p_USSMEMAConvStart		:= ADR(bConvStart);
	p_USSMEMAConvStop		:= ADR(bConvStop);
	p_USSMEMAUSB			:= ADR(bUSB);
	p_USSMEMATimer			:= ADR(bTimer);
	p_USSMEMAVirtual		:= ADR(bVirtual);

	(* Always Change If Project Change *)

END_PROGRAM
```

#### Act_InitGlobal.st - Change By Project
```iecst
(** 2019-04-09 **)
ACTION Act_InitGlobal:

	(* Always Change If Project Change *)

	//Pass Data To Link
	p_bLinkOpsRun ACCESS p_OpsRun;

	p_eLinkConvDir ACCESS p_NtParamProjConvDir;
	p_bLinkNtParamUSWidthChkPrep ACCESS p_NtParamUSWidthChkPrep;
	p_bLinkMcParamUSWidthChkEn ACCESS p_McParamUSWidthChkEn;
	p_bLinkDIUSWidthChkSen ACCESS p_DIUSWidthChkSen;

	//Pass Data To Internal Use
	p_udiRstErr ACCESS p_RstErrReset;
	p_bManual ACCESS p_UIMnlMod;
	p_tyParam ACCESS p_McParamUSSMEMAParam;
	p_diTransferInTO ACCESS p_McParamTranInErrDlyTm;
	p_bLeftSen ACCESS p_DIConvLftSen;
	p_bRightSen ACCESS p_DIConvRgtSen;
	p_bUBA ACCESS p_DIUBA;
	p_bUBAStat ACCESS p_DIUBAStat;
	p_bVirtualEn ACCESS p_UIVSMEMAUSEn;
	p_bUBAVirtual ACCESS p_UIVSMEMAUBA;
	p_bUBAStatVirtual ACCESS p_UIVSMEMAUBAStat;
	p_tRstDlyTm ACCESS p_NtParamUSSMEMARstDlyTm;
	p_tSigInChkTm ACCESS p_NtParamUSSMEMASigInChkTm;
	p_sProgNm ACCESS p_NtParamUSSMEMAProgNm;
	p_bNtSettingsLoadDone ACCESS p_StartupNtSettingsLoadDone;

	(* Always Change If Project Change *)

END_ACTION
```

#### InputRef_Link.var - Change By Project
```iecst
(*2019-04-09*)
(**)
VAR
	p_bLinkOpsRun : REFERENCE TO BOOL;
END_VAR
(**)
VAR
	p_eLinkConvDir : REFERENCE TO eConvDir;
	p_bLinkNtParamUSWidthChkPrep : REFERENCE TO BOOL;
	p_bLinkMcParamUSWidthChkEn : REFERENCE TO BOOL;
	p_bLinkDIUSWidthChkSen : REFERENCE TO BOOL;
END_VAR
```

#### Act_LinkAction.st - Change By Project
```iecst
(** 2019-04-09 **)
ACTION Act_LinkAction:

	IF p_bLinkOpsRun = TRUE THEN
		p_eAct ACCESS p_OpsInvertUSSMEMAAct;
	ELSIF p_bManual = TRUE THEN
		p_eAct ACCESS p_UIUSSMEMAAct;
	ELSE
		p_eAct ACCESS ADR(eAct);
	END_IF

END_ACTION
```
